// TwinCAT 3 PLC project TcBase
// Title: TcBase
// Company: TcBase
// Author: Giang Nguyen
// ProjectVersion: 0.1.2
// Description: Base library providing basic framework and design patterns.
// ProgramVersion: 3.1.4023.0
// libraries:
//   Base Interfaces,newest,System
//   Tc2_Standard, * (Beckhoff Automation GmbH)
//   Tc2_System, * (Beckhoff Automation GmbH)
//   Tc2_Utilities, * (Beckhoff Automation GmbH)
//   Tc3_DynamicMemory, * (Beckhoff Automation GmbH)
//   Tc3_Module, * (Beckhoff Automation GmbH)
//   TcUnit, * (www.tcunit.org)
// project tree:
//   Action/ FB_Action.TcPOU, FB_RunCyclicTasksAction.TcPOU, I_Action.TcIO
//   Action/Tests/ FB_ActionTestObject.TcPOU, FB_Action_Test.TcPOU, FB_ActivateAction.TcPOU
//   Collection/ FB_List.TcPOU, I_Collection.TcIO, I_Enumerable.TcIO, I_List.TcIO, Param_List.TcGVL
//   Collection/Tests/ FB_ListCapacity_Test.TcPOU, FB_List_Test.TcPOU
//   Context/ FB_Context.TcPOU, I_Context.TcIO
//   Cyclic Task/ I_CyclicTask.TcIO
//   / GVL_IntegerTypeBounds.TcGVL, TestTask.TcTTO
//   Helpers/ F_CompareObjects.TcPOU
//   Invocation Control/ FB_InvocationControl.TcPOU
//   Invocation Control/Tests/ FB_InvocationControlTestTask.TcPOU, FB_InvocationControl_Test.TcPOU
//   Object/ FB_LinkedObject.TcPOU, FB_Object.TcPOU, I_LinkedObject.TcIO, I_Object.TcIO
//   Object/Tests/ FB_DummyObject.TcPOU, FB_Object_Test.TcPOU
//   Observer Pattern/Abstraction/Actions/ FB_NotifyObserverAction.TcPOU
//   Observer Pattern/Abstraction/ FB_AbstractObservable.TcPOU, FB_AbstractObserver.TcPOU, I_Observable.TcIO, I_Observer.TcIO
//   Observer Pattern/ FB_Observable_BOOL.TcPOU, FB_Observable_LINT.TcPOU, FB_Observable_ULINT.TcPOU, FB_Observable_SINT.TcPOU, FB_Observable_DINT.TcPOU, FB_Observable_LWORD.TcPOU, FB_Observable_LREAL.TcPOU, FB_Observable_REAL.TcPOU, FB_Observable_INT.TcPOU, FB_Observable_USINT.TcPOU, FB_Observable_UDINT.TcPOU, FB_Observable_DWORD.TcPOU, FB_Observable_UINT.TcPOU, FB_Observable_BYTE.TcPOU, FB_Observable_WORD.TcPOU, FB_ObserverExt.TcPOU, FB_Observer_LINT.TcPOU, FB_Observer_ULINT.TcPOU, FB_Observer_SINT.TcPOU, FB_Observer_DINT.TcPOU, FB_Observer_LWORD.TcPOU, FB_Observer_LREAL.TcPOU, FB_Observer_REAL.TcPOU, FB_Observer_INT.TcPOU, FB_Observer_USINT.TcPOU, FB_Observer_UDINT.TcPOU, FB_Observer_DWORD.TcPOU, FB_Observer_UINT.TcPOU, FB_Observer_BOOL.TcPOU, FB_Observer_BYTE.TcPOU, FB_Observer_WORD.TcPOU
//   Observer Pattern/Tests/ FB_ObserverPattern_Test.TcPOU, FB_Observer_LREAL_.TcPOU
//   Programs/ Test.TcPOU
//   Restorable/ I_ObjectRestorer.TcIO, I_Restorable.TcIO
//   State Pattern/ FB_State.TcPOU, FB_StateMachine.TcPOU, I_State.TcIO, I_StateMachine.TcIO
//   State Pattern/Tests/ FB_StatePattern_Test.TcPOU
//   State Pattern/Tests/Test Subjects/ E_Season.TcDUT, FB_Autumn.TcPOU, FB_Default.TcPOU, FB_SeasonBase.TcPOU, FB_SeasonStateMachine.TcPOU, FB_Spring.TcPOU, FB_State1.TcPOU, FB_State2.TcPOU, FB_State3.TcPOU, FB_State4.TcPOU, FB_StateMachine1.TcPOU, FB_Summer.TcPOU, FB_Winter.TcPOU, FB_Year.TcPOU, I_SeasonControl.TcIO, I_SeasonState.TcIO
//   Task/Data Type/ E_TaskState.TcDUT
//   Task/ FB_Task.TcPOU, I_Task.TcIO, I_TaskStatus.TcIO

CONFIGURATION TcBase
    RESOURCE PLC ON TwinCAT3
        TASK TestTask(INTERVAL := T#10ms, PRIORITY := 1);
        PROGRAM Test WITH TestTask : Test;
    END_RESOURCE
END_CONFIGURATION

// ---- State Pattern/Tests/Test Subjects/E_Season.TcDUT
{attribute 'qualified_only'}
{attribute 'strict'}
{attribute 'to_string'}
TYPE E_Season :
(
    Autumn,
    Winter,
    Spring,
    Summer
);
END_TYPE

// ---- Task/Data Type/E_TaskState.TcDUT
{attribute 'qualified_only'}
{attribute 'strict'}
{attribute 'to_string'}
TYPE E_TaskState :
(
    Ready := 0,
    Busy,
    Error,
    Done
);
END_TYPE

// ---- Collection/Param_List.TcGVL
{attribute 'qualified_only'}
VAR_GLOBAL CONSTANT
    nDefaultCapacity: UDINT := 4;
    nMaxLength: UDINT := 16#7FEFFFFF;
END_VAR

// ---- GVL_IntegerTypeBounds.TcGVL
{attribute 'qualified_only'}
VAR_GLOBAL CONSTANT
    BYTE_UPPER_BOUND:       BYTE := 16#FF;
    WORD_UPPER_BOUND:       WORD := 16#FFFF;
    DWORD_UPPER_BOUND:      DWORD := 16#FFFF_FFFF;
    LWORD_UPPER_BOUND:      LWORD := 16#FFFF_FFFF_FFFF_FFFF;
    SINT_LOWER_BOUND:       SINT := TO_SINT(16#80);
    SINT_UPPER_BOUND:       SINT := 16#7F;
    USINT_UPPER_BOUND:      USINT := 16#FF;
    INT_LOWER_BOUND:        INT := TO_INT(16#8000);
    INT_UPPER_FOUND:        INT := 16#7FFF;
    UINT_UPPER_BOUND:       UINT := 16#FFFF;
    DINT_LOWER_BOUND:       DINT := TO_DINT(16#8000_0000);
    DINT_UPPER_BOUND:       DINT := 16#7FFF_FFFF;
    UDINT_UPPER_BOUND:      UDINT := 16#FFFF_FFFF;
    LINT_LOWER_BOUND:       LINT := TO_LINT(16#8000_0000_0000_0000);
    LINT_UPPER_BOUND:       LINT := 16#7FFF_FFFF_FFFF_FFFF;
    ULINT_UPPER_BOUND:      ULINT := 16#FFFF_FFFF_FFFF_FFFF;
END_VAR

// ---- Action/I_Action.TcIO
INTERFACE I_Action EXTENDS I_Object

METHOD Execute
VAR_INPUT
    ipObject: I_Object;
END_VAR
END_METHOD

END_INTERFACE

// ---- Collection/I_Collection.TcIO
INTERFACE I_Collection EXTENDS I_Enumerable

METHOD AddItem : DINT
// Returns the index to which the new object is added into the list,
// or -1  to indicate that the object was not inserted
VAR_INPUT
    ipObject:       I_Object;
END_VAR
END_METHOD

METHOD Clear
// Remove all items from the list
VAR_INPUT
END_VAR
END_METHOD

METHOD Contains : BOOL
// Determines whether the list contains the querried object
VAR_INPUT
    ipObject:       I_Object;
END_VAR
END_METHOD

METHOD CopyToArray : BOOL
// Copies the whole list to a compatible one-dimensional array,
// starting at a specified index
VAR_IN_OUT
    aDest:          ARRAY [*] OF I_Object;
END_VAR
VAR_INPUT
    nIdx:           DINT;
END_VAR
END_METHOD

PROPERTY nCount : UDINT
GET
END_GET
END_PROPERTY

METHOD Remove : BOOL
// Remove the first occurerence of a specific object from the list
VAR_INPUT
    ipObject:       I_Object;
END_VAR
END_METHOD

END_INTERFACE

// ---- Collection/I_Enumerable.TcIO
INTERFACE I_Enumerable EXTENDS I_Object

METHOD ForEach : I_Enumerable
VAR_INPUT
    ipAction: I_Action;
END_VAR
END_METHOD

END_INTERFACE

// ---- Collection/I_List.TcIO
INTERFACE I_List EXTENDS I_Collection, I_Enumerable

METHOD IndexOfItem : DINT
// Returns the zero-based index of the object if it was found in the list,
// otherwise returns -1
VAR_INPUT
    ipObject:       I_Object;
END_VAR
END_METHOD

METHOD Insert : BOOL
// Returns TRUE when object is inserted successfully, and FALSE otherwise
VAR_INPUT
    nIdx:       DINT; // Zero-based index at which object should be inserted
    ipObject:   I_Object; // Object to be inserted
END_VAR
END_METHOD

METHOD ItemAt : I_Object
VAR_INPUT
    nIdx:       DINT;
END_VAR
END_METHOD

METHOD LastIndexOf : DINT
VAR_INPUT
    ipObject:       I_Object;
END_VAR
END_METHOD

PROPERTY nCount : UDINT
GET
END_GET
END_PROPERTY

PROPERTY nItemSize : UDINT // Byte-size of each item
GET
END_GET
END_PROPERTY

METHOD RemoveAt : BOOL
// Remove an object at the specified index
VAR_INPUT
    nIdx:       DINT;
END_VAR
END_METHOD

END_INTERFACE

// ---- Context/I_Context.TcIO
INTERFACE I_Context EXTENDS I_Object

END_INTERFACE

// ---- Cyclic Task/I_CyclicTask.TcIO
INTERFACE I_CyclicTask EXTENDS __SYSTEM.IQueryInterface

METHOD Run
VAR_INPUT
END_VAR
END_METHOD

END_INTERFACE

// ---- Object/I_LinkedObject.TcIO
INTERFACE I_LinkedObject EXTENDS I_Object

PROPERTY ipContext : I_Context
GET
END_GET
END_PROPERTY

PROPERTY ipParent : I_LinkedObject
GET
END_GET
END_PROPERTY

END_INTERFACE

// ---- Object/I_Object.TcIO
INTERFACE I_Object EXTENDS __SYSTEM.IQueryInterface

METHOD Equals : BOOL
VAR_INPUT
    ipObject:       I_Object;
END_VAR
END_METHOD

PROPERTY nIdentity : ULINT
GET
END_GET
END_PROPERTY

PROPERTY sPath : STRING(MAX_STRING_LENGTH)
GET
END_GET
END_PROPERTY

END_INTERFACE

// ---- Observer Pattern/Abstraction/I_Observable.TcIO
INTERFACE I_Observable EXTENDS I_Object

METHOD Attach : BOOL
VAR_INPUT
    ipObserver:         I_Observer;
END_VAR
END_METHOD

(*Notify automatically on write access of observable value*)
PROPERTY bAutoNotify : BOOL
GET
END_GET
SET
END_SET
END_PROPERTY

(*Notify only when the value is actually changed*)
PROPERTY bNotifyWhenChanged : BOOL
GET
END_GET
SET
END_SET
END_PROPERTY

METHOD Detach : BOOL
VAR_INPUT
    ipObserver:         I_Observer;
END_VAR
END_METHOD

PROPERTY nDataSize : UDINT
GET
END_GET
END_PROPERTY

PROPERTY nObserverCount : UDINT
GET
END_GET
END_PROPERTY

METHOD NotifyAll : I_Observable
VAR_INPUT
END_VAR
END_METHOD

METHOD NotifyLast : I_Observable
VAR_INPUT
END_VAR
END_METHOD

PROPERTY nTypeClass : __SYSTEM.TYPE_CLASS
GET
END_GET
END_PROPERTY

METHOD ABSTRACT ValueChanged : BOOL
VAR_INPUT
END_VAR
END_METHOD

END_INTERFACE

// ---- Observer Pattern/Abstraction/I_Observer.TcIO
INTERFACE I_Observer EXTENDS I_Object

PROPERTY nTypeClass : __SYSTEM.TYPE_CLASS
GET
END_GET
END_PROPERTY

METHOD Update
VAR_INPUT
    anyVal:         ANY;
END_VAR
END_METHOD

METHOD UpdateP
VAR_INPUT
    pData:          POINTER TO BYTE;
    nTypeClass:     __SYSTEM.TYPE_CLASS;
    nSize:          UDINT;
END_VAR
END_METHOD

END_INTERFACE

// ---- Restorable/I_ObjectRestorer.TcIO
INTERFACE I_ObjectRestorer EXTENDS __SYSTEM.IQueryInterface

METHOD RestoreObject : I_ObjectRestorer
VAR_INPUT
    ipRestorable:           I_Restorable;
END_VAR
END_METHOD

END_INTERFACE

// ---- Restorable/I_Restorable.TcIO
INTERFACE I_Restorable EXTENDS __SYSTEM.IQueryInterface

METHOD Restore : I_Restorable
VAR_INPUT
END_VAR
END_METHOD

END_INTERFACE

// ---- State Pattern/I_State.TcIO
INTERFACE I_State EXTENDS I_Object, I_CyclicTask, I_Restorable

METHOD AssignStateMachine : BOOL
VAR_INPUT
    ipStateMachine:     I_StateMachine;
END_VAR
END_METHOD

PROPERTY ipStateMachine : I_StateMachine
GET
END_GET
END_PROPERTY

METHOD MakeOrphan
VAR_INPUT
END_VAR
END_METHOD

METHOD OnEntry
VAR_INPUT
END_VAR
END_METHOD

METHOD OnExit
VAR_INPUT
END_VAR
END_METHOD

END_INTERFACE

// ---- State Pattern/I_StateMachine.TcIO
INTERFACE I_StateMachine EXTENDS I_Object, I_CyclicTask, I_Restorable

METHOD AddState : BOOL
VAR_INPUT
    ipState:        I_State;
END_VAR
END_METHOD

METHOD ClearStates
VAR_INPUT
END_VAR
END_METHOD

METHOD Contains : BOOL
VAR_INPUT
    ipState:        I_State;
END_VAR
END_METHOD

PROPERTY ipPrevState : I_State
GET
END_GET
END_PROPERTY

PROPERTY ipState : I_State
GET
END_GET
END_PROPERTY

PROPERTY nStateCount : UDINT
GET
END_GET
END_PROPERTY

METHOD SetState : BOOL
VAR_INPUT
    newState:           I_State;
END_VAR
END_METHOD

METHOD StateAt : I_State
VAR_INPUT
    nIdx:       DINT; // Zero-based index to list of state
END_VAR
END_METHOD

END_INTERFACE

// ---- State Pattern/Tests/Test Subjects/I_SeasonControl.TcIO
INTERFACE INTERNAL I_SeasonControl EXTENDS __SYSTEM.IQueryInterface

PROPERTY StateAutumn : I_State
GET
END_GET
END_PROPERTY

PROPERTY StateSpring : I_State
GET
END_GET
END_PROPERTY

PROPERTY StateSummer : I_State
GET
END_GET
END_PROPERTY

PROPERTY StateWinter : I_State
GET
END_GET
END_PROPERTY

END_INTERFACE

// ---- State Pattern/Tests/Test Subjects/I_SeasonState.TcIO
INTERFACE INTERNAL I_SeasonState EXTENDS I_State

PROPERTY bRaining : BOOL
GET
END_GET
END_PROPERTY

PROPERTY bSnowing : BOOL
GET
END_GET
END_PROPERTY

PROPERTY bSunShining : BOOL
GET
END_GET
END_PROPERTY

PROPERTY bWindBlowing : BOOL
GET
END_GET
END_PROPERTY

METHOD ChangeToSummerTyres
VAR_INPUT
END_VAR
END_METHOD

METHOD ChangeToWinterTyres
VAR_INPUT
END_VAR
END_METHOD

PROPERTY eState : E_Season
GET
END_GET
END_PROPERTY

METHOD ABSTRACT NextSeason
VAR_INPUT
END_VAR
END_METHOD

PROPERTY nLeavesState : BYTE
GET
END_GET
END_PROPERTY

PROPERTY nTyresType : BYTE
GET
END_GET
END_PROPERTY

PROPERTY sState : STRING(MAX_STRING_LENGTH)
GET
END_GET
END_PROPERTY

END_INTERFACE

// ---- Task/I_Task.TcIO
INTERFACE I_Task EXTENDS I_Object, I_TaskStatus, I_Restorable

METHOD Abort : I_TaskStatus
VAR_INPUT
END_VAR
END_METHOD

METHOD Invoke : I_TaskStatus
VAR_INPUT
END_VAR
END_METHOD

END_INTERFACE

// ---- Task/I_TaskStatus.TcIO
INTERFACE I_TaskStatus EXTENDS __SYSTEM.IQueryInterface

PROPERTY bBusy : BOOL
GET
END_GET
END_PROPERTY

PROPERTY bDone : BOOL
GET
END_GET
END_PROPERTY

PROPERTY bError : BOOL
GET
END_GET
END_PROPERTY

PROPERTY bReady : BOOL
GET
END_GET
END_PROPERTY

END_INTERFACE

// ---- Programs/Test.TcPOU
PROGRAM Test
VAR
    fbObjectTest: FB_Object_Test;
    fbListTest: FB_List_Test;
    fbListEnsureCapacityTest: FB_ListCapacity_Test;
    fbCallCtrlTest: FB_InvocationControl_Test;
    fbObserverPatternTest: FB_ObserverPattern_Test;
    fbStatePatternTest: FB_StatePattern_Test;
    fbActionTest: FB_Action_Test;
END_VAR

TcUnit.RUN();

END_PROGRAM

// ---- Object/Tests/FB_Object_Test.TcPOU
{attribute 'reflection'}
FUNCTION_BLOCK INTERNAL FB_Object_Test EXTENDS TcUnit.FB_TestSuite
VAR
    fbPathTester: FB_DummyObject;
    _sTestPath: STRING(MAX_STRING_LENGTH) := CONCAT(_sPath, '.fbPathTester');

    {attribute 'instance-path'}
    {attribute 'noinit'}
    _sPath: STRING(MAX_STRING_LENGTH);
END_VAR

TestCompareObjectToSelfExpectTrue();
TestCompareTwoDifferentObjectsExpectFalse();
TestIdentityCorrectness();
TestPathCorrectness();

METHOD PRIVATE TestCompareObjectToSelfExpectTrue
VAR_INST
    fbObject1:      FB_DummyObject;
END_VAR
TcUnit.TEST('TestCompareObjectToSelfExpectTrue');

THIS^.AssertTrue(Condition := fbObject1.Equals(fbObject1),
                 Message := 'Failed when comparing two equal objects');

TcUnit.TEST_FINISHED();
END_METHOD

METHOD PRIVATE TestCompareTwoDifferentObjectsExpectFalse
VAR_INST
    fbObject1:      FB_DummyObject;
    fbObject2:      FB_DummyObject;
END_VAR
TcUnit.TEST('TestCompareTwoDifferentObjectsExpectFalse');

THIS^.AssertFalse(Condition := fbObject1.Equals(fbObject2),
                  Message := 'Failed when comparing two equal objects');

TcUnit.TEST_FINISHED();
END_METHOD

METHOD PRIVATE TestIdentityCorrectness
VAR_INST
    fbObject: FB_DummyObject;
END_VAR
TcUnit.TEST('TestIdentityCorrectness');

THIS^.AssertEquals_ULINT(Expected := ADR(fbObject),
                         Actual := fbObject.nIdentity,
                         Message := 'Object indentity is not true');

TcUnit.TEST_FINISHED();
END_METHOD

METHOD PRIVATE TestPathCorrectness
TcUnit.TEST('TestPathCorrectness');

THIS^.AssertEquals_STRING(Expected := THIS^._sTestPath,
                          Actual := THIS^.fbPathTester.sPath,
                          Message := 'Object path is not true');

TcUnit.TEST_FINISHED();
END_METHOD

END_FUNCTION_BLOCK

// ---- Object/Tests/FB_DummyObject.TcPOU
FUNCTION_BLOCK INTERNAL FB_DummyObject EXTENDS FB_Object
VAR_INPUT
END_VAR
VAR_OUTPUT
END_VAR
VAR
    _nTest: INT;
END_VAR

PROPERTY nTest : INT
GET
nTest := THIS^._nTest;
END_GET
SET
THIS^._nTest := nTest;
END_SET
END_PROPERTY

END_FUNCTION_BLOCK

// ---- Object/FB_Object.TcPOU
{attribute 'reflection'}
FUNCTION_BLOCK ABSTRACT FB_Object IMPLEMENTS I_Object
VAR
    _nIdentity:         ULINT;
    _ipSelf:            I_Object;

    {attribute 'instance-path'}
    {attribute 'noinit'}
    _sPath:             STRING(MAX_STRING_LENGTH);
END_VAR

METHOD Equals : BOOL
VAR_INPUT
    ipObject:       I_Object;
END_VAR
THIS^._ipSelf := THIS^;
Equals := ipObject = THIS^._ipSelf;
END_METHOD

METHOD FB_init : BOOL
VAR_INPUT
    bInitRetains:           BOOL; // if TRUE, the retain variables are initialized (warm start / cold start)
    bInCopyCode:            BOOL;  // if TRUE, the instance afterwards gets moved into the copy code (online change)
END_VAR
THIS^._nIdentity := ADR(THIS^);
THIS^._ipSelf := THIS^;
END_METHOD

PROPERTY nIdentity : ULINT
GET
THIS^._nIdentity := ADR(THIS^);
nIdentity := THIS^._nIdentity;
END_GET
END_PROPERTY

PROPERTY sPath : STRING(MAX_STRING_LENGTH)
GET
sPath := THIS^._sPath;
END_GET
END_PROPERTY

END_FUNCTION_BLOCK

// ---- Collection/Tests/FB_List_Test.TcPOU
FUNCTION_BLOCK INTERNAL FB_List_Test EXTENDS TcUnit.FB_TestSuite
VAR
END_VAR

TestAdd5DifferentItemsExpectAll5Added();
TestAdd5TimesSameObjectExpectAll5Copies();
TestAddNullInterfaceExpectNothingAdded();
TestClearEmptyListExpectSuccess();
TestClearNonEmptyListExpectSuccess();
TestContainsAddedObjectsExpectSuccess();
TestContainsNullObjectExpectFailure();
TestContainsNullObjectFromEmptyListExpectFailure();
TestCopyToArrayOfCompatibleSizeExpectSuccess();
TestCopyToArrayOfIncompatibleSizeExpectFailure();
TestCopyToArrayWithInvalidIndexExpectFailure();
TestEmptyListMustHaveNoItem();
TestForEachWithActivateActionExpectSuccess();
TestForEachWithCylicTaskActionExpectSuccess();
TestIndexOfItem();
TestInsertIntoEmptyListExpectSuccess();
TestInsertIntoListOfItemsExpectSuccess();
TestLastIndexOfListOfMixedDuplicatesAndUniques();
TestRemoveByIndexAndReAddItemExpectCorrectItemOrder();
TestRemoveByIndexFromEmptyListExpectFailure();
TestRemoveByIndexFromListOf5DifferentItemsExpectSuccess();
TestRemoveByIndexFromListOf5ItemsExpectConsistentContents();
TestRemoveByInvalidIndexFromListOfItemsExpectFailure();
TestRemoveInvalidItemFromListExpectFailure();
TestRemoveValidItemFromListExpectSuccess();
TestMeasureAddPerformanceWithVeryManyItemsAdded();

METHOD PRIVATE TestAdd5DifferentItemsExpectAll5Added
VAR_INST
    fbList: FB_List(0);

    aObject: ARRAY [1..5] OF FB_DummyObject;
    ipTmp: I_Object;
    ipCmp: I_Object;
    i: UDINT;
END_VAR
TcUnit.TEST('TestAdd5DifferentItemsExpectAll5Added');

FOR i := 1 TO SIZEOF(aObject)/SIZEOF(aObject[1]) DO
    THIS^.AssertEquals_DINT(Expected := TO_DINT(i - 1),
                            Actual := fbList.AddItem(aObject[i]),
                            Message := 'Failed to add object to list');
END_FOR

THIS^.AssertEquals_UDINT(Expected := SIZEOF(aObject)/SIZEOF(aObject[1]),
                         Actual := fbList.nCount,
                         Message := 'Unexpected number of items added to list');

FOR i := 1 TO SIZEOF(aObject)/SIZEOF(aObject[1]) DO
    ipTmp := fbList.ItemAt(TO_DINT(i - 1));
    ipCmp := aObject[i];
    THIS^.AssertTrue(Condition := ipTmp = ipCmp,
                     Message := CONCAT('Unexpected item at index ', TO_STRING(i)));
END_FOR

TcUnit.TEST_FINISHED();
END_METHOD

METHOD PRIVATE TestAdd5TimesSameObjectExpectAll5Copies
VAR_INST
    fbList: FB_List(0);

    nTimesToAdd: UDINT;
    fbObject: FB_DummyObject;
    ipTmp: I_Object;
    ipCmp: I_Object;
    i: UDINT;
END_VAR
TcUnit.TEST('TestAdd5TimesSameObjectExpectAll5Copies');

nTimesToAdd := 5;

FOR i := 1 TO nTimesToAdd DO
    THIS^.AssertEquals_DINT(Expected := TO_DINT(i - 1),
                            Actual := fbList.AddItem(fbObject),
                            Message := 'Failed to add object to list');
END_FOR

THIS^.AssertEquals_UDINT(Expected := nTimesToAdd,
                         Actual := fbList.nCount,
                         Message := 'Unexpected number of items added to list');

FOR i := 1 TO nTimesToAdd DO
    ipTmp := fbList.ItemAt(TO_DINT(i - 1));
    ipCmp := fbObject;
    THIS^.AssertTrue(Condition := ipTmp = ipCmp,
                     Message := 'Unexpected item added to list');
END_FOR

TcUnit.TEST_FINISHED();
END_METHOD

METHOD PRIVATE TestAddNullInterfaceExpectNothingAdded
VAR_INST
    fbList: FB_List(0);

    ipTmp: I_Object;
    i: UDINT;
END_VAR
TcUnit.TEST('TestAddNullInterfaceExpectNothingAdded');

FOR i := 1 TO 5 DO
    THIS^.AssertEquals_DINT(Expected := -1,
                            Actual := fbList.AddItem(ipTmp),
                            Message := 'Null item added to list');
END_FOR

THIS^.AssertEquals_UDINT(Expected := 0,
                         Actual := fbList.nCount,
                         Message := 'List has item(s) in it, but it should not');

TcUnit.TEST_FINISHED();
END_METHOD

METHOD PRIVATE TestClearEmptyListExpectSuccess
VAR_INST
    fbList: FB_List(0);
END_VAR
TcUnit.TEST('TestClearEmptyListExpectSuccess');

fbList.Clear();

THIS^.AssertEquals_UDINT(Expected := 0,
                         Actual := fbList.nCount,
                         Message := 'List should be empty');

TcUnit.TEST_FINISHED();
END_METHOD

METHOD PRIVATE TestClearNonEmptyListExpectSuccess
VAR_INST
    fbList: FB_List(0);

    aObject: ARRAY [1..5] OF FB_DummyObject;
    ipTmp: I_Object;
    i: UDINT;
END_VAR
TcUnit.TEST('TestClearNonEmptyListExpectSuccess');

FOR i := 1 TO SIZEOF(aObject)/SIZEOF(aObject[1]) DO
    fbList.AddItem(aObject[i]);
END_FOR

THIS^.AssertEquals_UDINT(Expected := SIZEOF(aObject)/SIZEOF(aObject[1]),
                         Actual := fbList.nCount,
                         Message := 'Unexpected number of items added to list');

fbList.Clear();

THIS^.AssertEquals_UDINT(Expected := 0,
                         Actual := fbList.nCount,
                         Message := 'List was not correctly cleared');

FOR i := 1 TO SIZEOF(aObject)/SIZEOF(aObject[1]) DO
    ipTmp := fbList.ItemAt(TO_DINT(i));
    THIS^.AssertTrue(Condition := ipTmp = 0,
                     Message := 'List was not correctly cleared');
END_FOR

TcUnit.TEST_FINISHED();
END_METHOD

METHOD PRIVATE TestContainsAddedObjectsExpectSuccess
VAR_INST
    fbList: FB_List(0);

    aObject: ARRAY [1..5] OF FB_DummyObject;

    ipNull: I_Object;
    i: UDINT;
END_VAR
TcUnit.TEST('TestContainsAddedObjectsExpectSuccess');

FOR i := 1 TO SIZEOF(aObject)/SIZEOF(aObject[1]) DO
    fbList.AddItem(aObject[i]);
END_FOR

FOR i := 1 TO SIZEOF(aObject)/SIZEOF(aObject[1]) DO
    THIS^.AssertTrue(Condition := fbList.Contains(aObject[i]),
                     Message := 'List does not contain added item');
END_FOR

THIS^.AssertFalse(Condition := fbList.Contains(ipNull),
                  Message := 'List should not contain null object');

TcUnit.TEST_FINISHED();
END_METHOD

METHOD PRIVATE TestContainsNullObjectExpectFailure
VAR_INST
    fbList: FB_List(0);

    ipNull: I_Object;
END_VAR
TcUnit.TEST('TestContainsNullObjectExpectFailure');

THIS^.AssertFalse(Condition := fbList.Contains(ipNull),
                  Message := 'List should not contain null object');

TcUnit.TEST_FINISHED();
END_METHOD

METHOD PRIVATE TestContainsNullObjectFromEmptyListExpectFailure
VAR_INST
    fbList: FB_List(0);

    aObject: ARRAY [1..5] OF FB_DummyObject;

    ipNull: I_Object;
    i: UDINT;
END_VAR
TcUnit.TEST('TestContainsNullObjectFromEmptyListExpectFailure');

FOR i := 1 TO SIZEOF(aObject)/SIZEOF(aObject[1]) DO
    fbList.AddItem(aObject[i]);
END_FOR

THIS^.AssertFalse(Condition := fbList.Contains(ipNull),
                  Message := 'List should not contain null object');

TcUnit.TEST_FINISHED();
END_METHOD

METHOD PRIVATE TestCopyToArrayOfCompatibleSizeExpectSuccess
VAR_INST
    fbList: FB_List(0);
    nObjectCount: UDINT;
    aSrcObject: ARRAY [1..10] OF FB_DummyObject;
    aDestObject: ARRAY [1..10] OF I_Object;
    aDestObject2: ARRAY [1..30] OF I_Object;
    i: UDINT;
    ipObject: I_Object;

END_VAR
TcUnit.TEST('TestCopyToArrayOfCompatibleSizeExpectSuccess');

nObjectCount := SIZEOF(aSrcObject)/SIZEOF(aSrcObject[1]);
FOR i := 1 TO nObjectCount DO
    fbList.AddItem(aSrcObject[i]);
END_FOR

// Copy to same size array without offset
THIS^.AssertTrue(Condition := fbList.CopyToArray(aDestObject, 1),
                 Message := 'Failed to copy list to array of same size');

FOR i := 1 TO nObjectCount DO
    ipObject := aSrcObject[i];
    THIS^.AssertTrue(Condition := ipObject = aDestObject[i],
                     Message := 'Expected the same object after in array after copying from list');
END_FOR

// Copy to bigger array with offset
THIS^.AssertTrue(Condition := fbList.CopyToArray(aDestObject2, 14),
                 Message := 'Failed to copy list to array with bigger size');

FOR i := 1 TO nObjectCount DO
    ipObject := aSrcObject[i];
    THIS^.AssertTrue(Condition := ipObject = aDestObject2[i + 13],
                     Message := 'Expected the same object after in array after copying from list');
END_FOR

TcUnit.TEST_FINISHED();
END_METHOD

METHOD PRIVATE TestCopyToArrayOfIncompatibleSizeExpectFailure
VAR_INST
    fbList: FB_List(0);
    nObjectCount: UDINT;
    aSrcObject: ARRAY [1..10] OF FB_DummyObject;
    aDestObject: ARRAY [1..5] OF I_Object;
    i: UDINT;
END_VAR
TcUnit.TEST('TestCopyToArrayOfIncompatibleSizeExpectFailure');

nObjectCount := SIZEOF(aSrcObject)/SIZEOF(aSrcObject[1]);
FOR i := 1 TO nObjectCount DO
    fbList.AddItem(aSrcObject[i]);
END_FOR

THIS^.AssertFalse(Condition := fbList.CopyToArray(aDestObject, 1),
                  Message := 'Failed to copy list to array of same size');

FOR i := 1 TO SIZEOF(aDestObject)/SIZEOF(aDestObject[1]) DO
    THIS^.AssertTrue(Condition := aDestObject[i] = 0,
                     Message := 'Array should be "empty" after copying due to being smaller than list');
END_FOR

TcUnit.TEST_FINISHED();
END_METHOD

METHOD PRIVATE TestCopyToArrayWithInvalidIndexExpectFailure
VAR_INST
    fbList: FB_List(0);
    nObjectCount: UDINT;
    aSrcObject: ARRAY [1..10] OF FB_DummyObject;
    aDestObject: ARRAY [1..10] OF I_Object;
    aDestObject2: ARRAY [1..30] OF I_Object;
    i: UDINT;

END_VAR
TcUnit.TEST('TestCopyToArrayWithInvalidIndexExpectFailure');

nObjectCount := SIZEOF(aSrcObject)/SIZEOF(aSrcObject[1]);
FOR i := 1 TO nObjectCount DO
    fbList.AddItem(aSrcObject[i]);
END_FOR

// Copy to same size array
THIS^.AssertFalse(Condition := fbList.CopyToArray(aDestObject, 2),
                  Message := 'List should not copy items to array using invalid index');

FOR i := 1 TO nObjectCount DO
    THIS^.AssertTrue(Condition := 0 = aDestObject[i],
                     Message := 'Array should be "empty" after copying due to being smaller than list');
END_FOR

// Copy to bigger array
THIS^.AssertFalse(Condition := fbList.CopyToArray(aDestObject2, 22),
                  Message := 'List should not copy items to array using invalid index');

FOR i := 1 TO nObjectCount DO
    THIS^.AssertTrue(Condition := 0 = aDestObject2[i + 13],
                     Message := 'Array should be "empty" after copying due to being smaller than list');
END_FOR

THIS^.AssertFalse(Condition := fbList.CopyToArray(aDestObject2, 0),
                  Message := 'List should not copy items to array using invalid index');

FOR i := 1 TO nObjectCount DO
    THIS^.AssertTrue(Condition := 0 = aDestObject2[i + 13],
                     Message := 'Array should be "empty" after copying due to being smaller than list');
END_FOR

TcUnit.TEST_FINISHED();
END_METHOD

METHOD PRIVATE TestEmptyListMustHaveNoItem
VAR_INST
    fbList:     FB_List(0);
END_VAR
TcUnit.TEST('TestEmptyListMustHaveNoItem');

THIS^.AssertEquals_UDINT(Expected := 0,
                         Actual := fbList.nCount,
                         Message := 'Empty list must not have any item(s)');

TcUnit.TEST_FINISHED();
END_METHOD

METHOD PRIVATE TestForEachWithActivateActionExpectSuccess
VAR_INST
    i: UDINT;
    fbList: FB_List(0);
    aObject: ARRAY [1..10] OF FB_ActionTestObject;
    fbActivateObjects: FB_ActivateAction;
END_VAR
TcUnit.TEST('TestForEachWithActivateActionExpectSuccess');

FOR i := 1 TO SIZEOF(aObject)/SIZEOF(aObject[1]) DO
    fbList.AddItem(aObject[i]);
END_FOR

fbList.ForEach(fbActivateObjects.Inputs(TRUE));

FOR i := 1 TO SIZEOF(aObject)/SIZEOF(aObject[1]) DO
     THIS^.AssertTrue(Condition := aObject[1].bIsActivated,
                      Message := 'Failed to activate object(s)');
END_FOR

TcUnit.TEST_FINISHED();
END_METHOD

METHOD PRIVATE TestForEachWithCylicTaskActionExpectSuccess
VAR_INST
    nCyclesToRun: UDINT := 5;
    nCounter: UDINT := 0;
    i: UDINT;
    fbList: FB_List(0);
    aObject: ARRAY [1..10] OF FB_ActionTestObject;
    fbRunCyclicTask: FB_RunCyclicTasksAction;
END_VAR
TcUnit.TEST('TestForEachWithCylicTaskActionExpectSuccess');

IF nCounter = 0 THEN
    FOR i := 1 TO SIZEOF(aObject)/SIZEOF(aObject[1]) DO
        fbList.AddItem(aObject[i]);
    END_FOR
END_IF

fbList.ForEach(fbRunCyclicTask);
nCounter := nCounter + 1;

IF nCyclesToRun = nCounter THEN
    FOR i := 1 TO SIZEOF(aObject)/SIZEOF(aObject[1]) DO
        THIS^.AssertEquals_UDINT(Expected := nCyclesToRun,
                                 Actual := aObject[i].nCounter,
                                 Message := 'Unexpected counter value of cyclic object');
    END_FOR
    TcUnit.TEST_FINISHED();
END_IF
END_METHOD

METHOD PRIVATE TestIndexOfItem
VAR_INST
    fbList: FB_List(0);

    aObject: ARRAY [1..10] OF FB_DummyObject;
    fbObject1: FB_DummyObject;
    fbObject2: FB_DummyObject;
    fbObject3: FB_DummyObject;

    ipNull: I_Object;
    i: UDINT;
END_VAR
TcUnit.TEST('TestIndexQuerryCorrectness');

FOR i := 1 TO SIZEOF(aObject)/SIZEOF(aObject[1]) DO
    fbList.AddItem(aObject[i]);
END_FOR

FOR i := 1 TO SIZEOF(aObject)/SIZEOF(aObject[1]) DO
    THIS^.AssertEquals_DINT(Expected := TO_DINT(i - 1),
                            Actual := fbList.IndexOfItem(aObject[i]),
                            Message := 'Unexpected index of added item');
END_FOR

fbList.Clear();

FOR i := 1 TO SIZEOF(aObject)/SIZEOF(aObject[1]) DO
    THIS^.AssertEquals_DINT(Expected := -1,
                            Actual := fbList.IndexOfItem(aObject[i]),
                            Message := 'Item still found from list even though it has been cleared');
END_FOR

THIS^.AssertEquals_DINT(Expected := -1,
                        Actual := fbList.IndexOfItem(ipNull),
                        Message := 'Invalid result when querying index of a null item');

fbList.AddItem(fbObject1);
fbList.AddItem(fbObject3);
fbList.AddItem(fbObject1);
fbList.AddItem(fbObject2);
fbList.AddItem(fbObject2);

THIS^.AssertEquals_DINT(Expected := 0,
                        Actual := fbList.IndexOfItem(fbObject1),
                        Message := 'IndexOfItem() should return the index of the first match if there are multiple copies');
THIS^.AssertEquals_DINT(Expected := 1,
                        Actual := fbList.IndexOfItem(fbObject3),
                        Message := 'IndexOfItem() should return the index of the first match if there are multiple copies');
THIS^.AssertEquals_DINT(Expected := 3,
                        Actual := fbList.IndexOfItem(fbObject2),
                        Message := 'IndexOfItem() should return the index of the first match if there are multiple copies');


TcUnit.TEST_FINISHED();
END_METHOD

METHOD PRIVATE TestInsertIntoEmptyListExpectSuccess
VAR_INST
    fbList: FB_List(0);

    aObject: ARRAY [1..10] OF FB_DummyObject;
    aInsPos: ARRAY [1..10] OF DINT;
    ipTmp: I_Object;
    ipCmp: I_Object;

    i: UDINT;
END_VAR
TcUnit.TEST('TestInsertIntoEmptyListExpectSuccess');

FOR i := 1 TO SIZEOF(aObject)/SIZEOF(aObject[1]) DO
    IF i = 4 THEN
        aInsPos[i] := 0;
    ELSIF i = 8 THEN
        aInsPos[i] := 4;;
    ELSIF i = 10 THEN
        aInsPos[i] := 1;
    ELSE
        aInsPos[i] := TO_DINT(i - 1);
    END_IF

    THIS^.AssertTrue(Condition := fbList.Insert(nIdx := aInsPos[i], aObject[i]),
                     Message := 'Could not insert item to list');

    ipTmp := fbList.ItemAt(aInsPos[i]);
    ipCmp := aObject[i];
    THIS^.AssertTrue(Condition := ipTmp = ipCmp,
                     Message := 'Added item is not at the expected index');
END_FOR

THIS^.AssertEquals_UDINT(Expected := SIZEOF(aObject)/SIZEOF(aObject[1]),
                         Actual := fbList.nCount,
                         Message := 'Unexpected number of items inserted to list');

FOR i := 1 TO SIZEOF(aObject)/SIZEOF(aObject[1]) DO
    THIS^.AssertTrue(Condition := fbList.Contains(aObject[i]),
                     Message := 'List does not contain inserted item');
END_FOR

TcUnit.TEST_FINISHED();
END_METHOD

METHOD PRIVATE TestInsertIntoListOfItemsExpectSuccess
VAR_INST
    fbList: FB_List(0);

    aObject: ARRAY [1..10] OF FB_DummyObject;
    aObjectToInsert: ARRAY [1..3] OF FB_DummyObject;
    aInsPos: ARRAY [1..3] OF DINT;
    ipTmp: I_Object;
    ipCmp: I_Object;

    i: UDINT;
END_VAR
TcUnit.TEST('TestInsertIntoListOfItemsExpectSuccess');

{region "Insert to head, end, and middle"}
FOR i := 1 TO SIZEOF(aObject)/SIZEOF(aObject[1]) DO
    fbList.AddItem(aObject[i]);
END_FOR

aInsPos[1] := 0;
aInsPos[2] := TO_DINT(fbList.nCount + 1);
aInsPos[3] := 3;

FOR i := 1 TO SIZEOF(aInsPos)/SIZEOF(aInsPos[1]) DO
    THIS^.AssertTrue(Condition := fbList.Insert(aInsPos[i], aObjectToInsert[i]),
                     Message := 'Failed to insert item into list');

    ipTmp := fbList.ItemAt(aInsPos[i]);
    ipCmp := aObjectToInsert[i];
    THIS^.AssertTrue(Condition := ipTmp = ipCmp,
                     Message := 'Added item is not at the expected index');
END_FOR

THIS^.AssertEquals_UDINT(Expected := SIZEOF(aObject)/SIZEOF(aObject[1])
                                     + SIZEOF(aObjectToInsert)/SIZEOF(aObjectToInsert[1]),
                         Actual := fbList.nCount,
                         Message := 'Unexpected number of items inserted to list');

FOR i := 1 TO SIZEOF(aObject)/SIZEOF(aObject[1]) DO
    THIS^.AssertTrue(Condition := fbList.Contains(aObject[i]),
                     Message := 'List does not contain inserted item');
END_FOR

FOR i := 1 TO SIZEOF(aObjectToInsert)/SIZEOF(aObjectToInsert[1]) DO
    THIS^.AssertTrue(Condition := fbList.Contains(aObjectToInsert[i]),
                     Message := 'List does not contain inserted item');
END_FOR
{endregion}

fbList.Clear();

{region "Insert to middle"}
FOR i := 1 TO SIZEOF(aObject)/SIZEOF(aObject[1]) DO
    fbList.AddItem(aObject[i]);
END_FOR

aInsPos[1] := 8;
aInsPos[2] := 5;
aInsPos[3] := 1;

FOR i := 1 TO SIZEOF(aInsPos)/SIZEOF(aInsPos[1]) DO
    THIS^.AssertTrue(Condition := fbList.Insert(aInsPos[i], aObjectToInsert[i]),
                     Message := 'Failed to insert item into list');

    ipTmp := fbList.ItemAt(aInsPos[i]);
    ipCmp := aObjectToInsert[i];
    THIS^.AssertTrue(Condition := ipTmp = ipCmp,
                     Message := 'Added item is not at the expected index');
END_FOR

THIS^.AssertEquals_UDINT(Expected := SIZEOF(aObject)/SIZEOF(aObject[1])
                                     + SIZEOF(aObjectToInsert)/SIZEOF(aObjectToInsert[1]),
                         Actual := fbList.nCount,
                         Message := 'Unexpected number of items inserted to list');

FOR i := 1 TO SIZEOF(aObject)/SIZEOF(aObject[1]) DO
    THIS^.AssertTrue(Condition := fbList.Contains(aObject[i]),
                     Message := 'List does not contain inserted item');
END_FOR

FOR i := 1 TO SIZEOF(aObjectToInsert)/SIZEOF(aObjectToInsert[1]) DO
    THIS^.AssertTrue(Condition := fbList.Contains(aObjectToInsert[i]),
                     Message := 'List does not contain inserted item');
END_FOR
{endregion}

TcUnit.TEST_FINISHED();
END_METHOD

METHOD PRIVATE TestLastIndexOfListOfMixedDuplicatesAndUniques
VAR_INST
    fbList: FB_List(0);

    aObject: ARRAY [1..5] OF FB_DummyObject;
    aAddOrder: ARRAY[1..20] OF I_Object;
    aExpLastIdx: ARRAY [1..5] OF DINT;
    nIdx: UDINT;
    nObjectCount: UDINT;
    nTimesToAdd: UDINT;
    i: UDINT;
    fbRand: DRAND := (Seed := 128);
    sMessage: STRING(255);
END_VAR
TcUnit.TEST('TestLastIndexOfListOfMixedDuplicatesAndUniques');

nObjectCount := SIZEOF(aObject)/SIZEOF(aObject[1]);
nTimesToAdd := SIZEOF(aAddOrder)/SIZEOF(aAddOrder[1]);

FOR i := 1 TO nTimesToAdd DO
    fbRand();
    nIdx := TO_UDINT(fbRand.Num*(nObjectCount - 1)) + 1;
    aAddOrder[i] := aObject[nIdx];

    IF aExpLastIdx[nIdx] < TO_DINT(i) THEN
        aExpLastIdx[nIdx] := TO_DINT(i);
    END_IF
END_FOR

FOR i := 1 TO nTimesToAdd DO
    fbList.AddItem(aAddOrder[i]);
END_FOR

FOR i := 1 TO nObjectCount DO
    sMessage := Tc2_Standard.CONCAT('Unexpected last index of object at idx ', TO_STRING(i));
    THIS^.AssertEquals_DINT(Expected := aExpLastIdx[i] - 1,
                            Actual := fbList.LastIndexOf(aObject[i]),
                            Message := sMessage);
END_FOR

TcUnit.TEST_FINISHED();
END_METHOD

METHOD PRIVATE TestMeasureAddPerformanceWithVeryManyItemsAdded
VAR_INST
    fbList: FB_List(0);
    fbObject: FB_DummyObject;
    fbProfiler: Tc2_Utilities.Profiler;

    nTimesToAdd: UDINT := 100000;
    i: UDINT;
    stProfileData: Tc2_Utilities.PROFILERSTRUCT;
    sMsg: STRING(255);
END_VAR
IF TcUnit.TEST_ORDERED('TestMeasureAddPerformanceWithVeryManyItemsAdded') THEN
    IF nTimesToAdd > 0 THEN
        fbProfiler(START := TRUE, RESET := TRUE);
        FOR i := 1 TO nTimesToAdd DO
            fbList.AddItem(fbObject);
        END_FOR

        THIS^.AssertEquals_UDINT(Expected := TO_UDINT(nTimesToAdd),
                                 Actual := fbList.nCount,
                                 Message := 'Unexpected number of items added to list');

        fbProfiler(START := FALSE);
        stProfileData := fbProfiler.DATA;

        sMsg := 'Took ';
        sMsg := CONCAT(sMsg, TO_STRING(stProfileData.LastExecTime));
        sMsg := CONCAT(sMsg, 'us to add ');
        sMsg := CONCAT(sMsg, TO_STRING(nTimesToAdd));
        sMsg := CONCAT(sMsg, ' item(s) to list. ');
        sMsg := CONCAT(sMsg, 'On average ');
        sMsg := CONCAT(sMsg, TO_STRING(TO_LREAL(fbProfiler.DATA.AverageExecTime)/TO_LREAL(nTimesToAdd)));
        sMsg := CONCAT(sMsg, 'us');
        sMsg := CONCAT(sMsg, ' per item');

        Tc2_System.ADSLOGSTR(msgCtrlMask := Tc2_System.ADSLOG_MSGTYPE_ERROR,
                             msgFmtStr := sMsg,
                             strArg := '');
    END_IF

    TcUnit.TEST_FINISHED();
END_IF
END_METHOD

METHOD PRIVATE TestRemoveByIndexAndReAddItemExpectCorrectItemOrder
VAR_INST
    fbList: FB_List(0);
    aObject: ARRAY [1..5] OF FB_DummyObject;
    aIdx: ARRAY [1..5] OF UDINT
        := [3, 2, 4, 5, 1];
    nArraySize: UDINT;
    i: UDINT;
    j: UDINT;
END_VAR
TcUnit.TEST('TestRemoveByIndexAndReAddItemExpectCorrectItemOrder');
nArraySize := SIZEOF(aObject)/SIZEOF(aObject[1]);

FOR i := 1 TO nArraySize DO
    fbList.AddItem(aObject[i]);
END_FOR

FOR i := 1 TO nArraySize DO
    fbList.RemoveAt(fbList.IndexOfItem(aObject[aIdx[i]]));
    fbList.AddItem(aObject[aIdx[i]]);
END_FOR

FOR i := 1 TO nArraySize DO
    THIS^.AssertTrue(Condition := fbList.ItemAt(TO_DINT(i) - 1).Equals(aObject[aIdx[i]]),
                     Message := CONCAT('Unexpected item found at ', TO_STRING(i - 1)));
END_FOR

TcUnit.TEST_FINISHED();
END_METHOD

METHOD PRIVATE TestRemoveByIndexFromEmptyListExpectFailure
VAR_INST
    fbList: FB_List(0);

    aIdx: ARRAY[1..10] OF DINT := 
        [0, 1, 2, 3, 4, 5, 6, 7, 8, 9];

    i: UDINT;
END_VAR
TcUnit.TEST('TestRemoveByIndexFromEmptyListExpectFailure');

FOR i := 1 TO SIZEOF(aIdx)/SIZEOF(aIdx[1]) DO
    THIS^.AssertFalse(Condition := fbList.RemoveAt(aIdx[i]),
                      Message := 'Empty list should not have any item to be removed');
END_FOR

TcUnit.TEST_FINISHED();
END_METHOD

METHOD PRIVATE TestRemoveByIndexFromListOf5DifferentItemsExpectSuccess
VAR_INST
    fbList: FB_List(0);
    aObject: ARRAY [1..5] OF FB_DummyObject;

    nArraySize: UDINT;
    i: UDINT;
END_VAR
TcUnit.TEST('TestRemoveItemFromListOf5DifferentItemsExpectSuccess');
nArraySize := SIZEOF(aObject)/SIZEOF(aObject[1]);

// Remove from last to first
FOR i := 1 TO nArraySize DO
    fbList.AddItem(aObject[i]);
END_FOR

FOR i := 1 TO nArraySize DO
    THIS^.AssertTrue(Condition := fbList.RemoveAt(TO_DINT(nArraySize - i)),
                     Message := 'Could not remove added item');

    THIS^.AssertEquals_UDINT(Expected := nArraySize - i,
                             Actual := fbList.nCount,
                             Message := 'Unexpected number of items after removal');
END_FOR

// Remove from first
FOR i := 1 TO nArraySize DO
    fbList.AddItem(aObject[i]);
END_FOR

FOR i := 1 TO nArraySize DO
    THIS^.AssertTrue(Condition := fbList.RemoveAt(0),
                     Message := 'Could not remove added item');

    THIS^.AssertEquals_UDINT(Expected := nArraySize - i,
                             Actual := fbList.nCount,
                             Message := 'Unexpected number of items after removal');
END_FOR

// Remove from middle to first
FOR i := 1 TO nArraySize DO
    fbList.AddItem(aObject[i]);
END_FOR

FOR i := 1 TO nArraySize DO
    THIS^.AssertTrue(Condition := fbList.RemoveAt(MAX(0, 3 - TO_DINT(i))),
                     Message := 'Could not remove added item');

    THIS^.AssertEquals_UDINT(Expected := nArraySize - i,
                             Actual := fbList.nCount,
                             Message := 'Unexpected number of items after removal');
END_FOR

TcUnit.TEST_FINISHED();
END_METHOD

METHOD PRIVATE TestRemoveByIndexFromListOf5ItemsExpectConsistentContents
VAR_INST
    fbList: FB_List(0);
    aObject: ARRAY [1..5] OF FB_DummyObject;
    nArraySize: UDINT;
    i: UDINT;
    j: UDINT;
END_VAR
TcUnit.TEST('TestRemoveByIndexFromListOf5ItemsExpectConsistentContents');
nArraySize := SIZEOF(aObject)/SIZEOF(aObject[1]);

FOR i := 1 TO nArraySize DO
    fbList.AddItem(aObject[i]);
END_FOR

FOR i := 1 TO nArraySize DO
    fbList.RemoveAt(0);

    // After every removal, we check that the content of the list is correct
    IF fbList.nCount > 0 THEN
        FOR j := 0 TO fbList.nCount - 1 DO
            THIS^.AssertTrue(Condition := fbList.ItemAt(TO_DINT(j)).Equals(aObject[i + j + 1]),
                             Message := 'Unexpected list contents after removing item');
        END_FOR
    END_IF
END_FOR

TcUnit.TEST_FINISHED();
END_METHOD

METHOD PRIVATE TestRemoveByInvalidIndexFromListOfItemsExpectFailure
VAR_INST
    fbList: FB_List(0);

    aIdx: ARRAY[1..10] OF DINT := 
        [-1, 5, 6, 7, 10, -10, -3, -4, -2, 9];
    aObject: ARRAY [1..5] OF FB_DummyObject;

    i: UDINT;
END_VAR
TcUnit.TEST('TestRemoveByInvalidIndexFromListOfItemsExpectFailure');

FOR i := 1 TO SIZEOF(aObject)/SIZEOF(aObject[1]) DO
    fbList.AddItem(aObject[i]);
END_FOR

FOR i := 1 TO SIZEOF(aIdx)/SIZEOF(aIdx[1]) DO
    THIS^.AssertFalse(Condition := fbList.RemoveAt(aIdx[i]),
                      Message := 'Removing item with out-of-bound index should not succeed');
END_FOR

THIS^.AssertEquals_UDINT(Expected := 5,
                         Actual := fbList.nCount,
                         Message := 'Item(s) were successfully removed from list with out-of-bound index');

TcUnit.TEST_FINISHED();
END_METHOD

METHOD PRIVATE TestRemoveInvalidItemFromListExpectFailure
VAR_INST
    fbList: FB_List(0);

    aObject: ARRAY [1..10] OF FB_DummyObject;
    ipNull: I_Object;
    fbObject: FB_DummyObject;

    i: UDINT;
END_VAR
TcUnit.TEST('TestRemoveInvalidItemFromListExpectFailure');

FOR i := 1 TO SIZEOF(aObject)/SIZEOF(aObject[1]) DO
    fbList.AddItem(aObject[i]);
END_FOR

THIS^.AssertFalse(Condition := fbList.Remove(ipNull),
                  Message := 'Unexpectedly removed a null item');

THIS^.AssertFalse(Condition := fbList.Remove(fbObject),
                  Message := 'List should not be able to remove item it does not contain');

THIS^.AssertEquals_UDINT(Expected := SIZEOF(aObject)/SIZEOF(aObject[1]),
                         Actual := fbList.nCount,
                         Message := 'Unexpected number of items after invalid removal');

FOR i := 1 TO SIZEOF(aObject)/SIZEOF(aObject[1]) DO
    THIS^.AssertTrue(Condition := fbList.Remove(aObject[i]),
                     Message := 'Could not remove added item');

    THIS^.AssertFalse(Condition := fbList.Remove(aObject[i]),
                      Message := 'Removed item was unexpectedly removed twice');

    THIS^.AssertEquals_UDINT(Expected := SIZEOF(aObject)/SIZEOF(aObject[1]) - i,
                             Actual := fbList.nCount,
                             Message := 'Unexpected number of items after removal');
END_FOR

TcUnit.TEST_FINISHED();
END_METHOD

METHOD PRIVATE TestRemoveValidItemFromListExpectSuccess
VAR_INST
    fbList: FB_List(0);

    aObject: ARRAY [1..10] OF FB_DummyObject;

    i: UDINT;
END_VAR
TcUnit.TEST('TestRemoveValidItemFromListExpectSuccess');

FOR i := 1 TO SIZEOF(aObject)/SIZEOF(aObject[1]) DO
    fbList.AddItem(aObject[i]);
END_FOR

FOR i := 1 TO SIZEOF(aObject)/SIZEOF(aObject[1]) DO
    THIS^.AssertTrue(Condition := fbList.Remove(aObject[i]),
                     Message := 'Could not remove added item');

    THIS^.AssertEquals_UDINT(Expected := SIZEOF(aObject)/SIZEOF(aObject[1]) - i,
                             Actual := fbList.nCount,
                             Message := 'Unexpected number of items after removal');
END_FOR

TcUnit.TEST_FINISHED();
END_METHOD

END_FUNCTION_BLOCK

// ---- Collection/FB_List.TcPOU
FUNCTION_BLOCK FB_List EXTENDS FB_Object IMPLEMENTS I_List
VAR
    fbMemMan:       FB_DynMem_Manager;
    fbBuffer:       FB_DynMem_Buffer(ipMemMan := fbMemMan);
    _nCount:        UDINT;
END_VAR

METHOD AddItem : DINT
VAR_INPUT
    ipObject:       I_Object;
END_VAR
IF ipObject = 0 THEN
    AddItem := -1;
    RETURN;
END_IF

IF THIS^.IsFull() THEN
    AddItem := -1;
    RETURN;
END_IF

IF THIS^.nCount = THIS^.nCapacity THEN
    THIS^.EnsureCapacity(THIS^.nCount + 1);
END_IF

THIS^._nCount := THIS^._nCount + 1;
THIS^.WriteToBuffer(nIdx := THIS^.nLastIdx, ipObject := ipObject);
AddItem := THIS^.nLastIdx;
END_METHOD

METHOD Clear
THIS^.fbBuffer.Resize(nSize := 0,
                      bPreserve := FALSE,
                      bReset := TRUE);

THIS^._nCount := 0;
END_METHOD

METHOD Contains : BOOL
VAR_INPUT
    ipObject:       I_Object;
END_VAR
VAR
    i:              DINT;
    ipTmp:          I_Object;
END_VAR
IF ipObject = 0 THEN
    RETURN;
END_IF

FOR i := 0 TO THIS^.nLastIdx DO
    IF F_CompareObjects(ipObject, THIS^.ItemAt(i)) THEN
        Contains := TRUE;
        RETURN;
    END_IF
END_FOR
END_METHOD

METHOD CopyToArray : BOOL
// Copies the whole list to a compatible one-dimensional array,
// starting at a specified index
VAR_IN_OUT
    aDest:          ARRAY [*] OF I_Object;
END_VAR
VAR_INPUT
    nIdx:           DINT;
END_VAR
VAR
    nLowerBnd:      DINT;
    nUpperBnd:      DINT;
    i:              DINT;
END_VAR
// Nothing to copy
IF THIS^.nCount = 0 THEN
    RETURN;
END_IF

nLowerBnd := LOWER_BOUND(aDest, 1);
nUpperBnd := UPPER_BOUND(aDest, 1);

// Invalid index given
IF nIdx < nLowerBnd OR_ELSE nUpperBnd < nIdx THEN
    RETURN;
END_IF

// Array not big enough
IF TO_UDINT(nUpperBnd - nIdx + 1) < THIS^.nCount THEN
    RETURN;
END_IF

Tc2_System.MEMCPY(destAddr := ADR(aDest[nIdx]),
                  srcAddr := THIS^.pBuffer,
                  n := THIS^.nCount*THIS^.nItemSize);

CopyToArray := TRUE;
END_METHOD

METHOD PRIVATE EnsureCapacity : BOOL
VAR_INPUT
    nMin: UDINT;
END_VAR
VAR
    nNewCapacity: UDINT;
END_VAR
IF THIS^.nCapacity > nMin THEN
    RETURN;
END_IF

nNewCapacity := SEL(THIS^.nCapacity = 0, THIS^.nCapacity * 2, Param_List.nDefaultCapacity);
nNewCapacity := LIMIT(nMin, nNewCapacity, Param_List.nMaxLength);

EnsureCapacity := THIS^.fbBuffer.Resize(nSize := nNewCapacity*THIS^.nItemSize,
                                        bPreserve := TRUE,
                                        bReset := FALSE);
END_METHOD

METHOD FB_init : BOOL
VAR_INPUT
    bInitRetains:   BOOL; // if TRUE, the retain variables are initialized (warm start / cold start)
    bInCopyCode:    BOOL;  // if TRUE, the instance afterwards gets moved into the copy code (online change)
    nCapacity:      UDINT;
END_VAR
THIS^.fbBuffer.CreateBuffer(nSize := nCapacity*THIS^.nItemSize,
                            bReset := TRUE);
END_METHOD

METHOD ForEach : I_Enumerable
VAR_INPUT
    ipAction: I_Action;
END_VAR
VAR
    i: DINT;
END_VAR
ForEach := THIS^;

IF THIS^.nCount = 0 OR_ELSE ipAction = 0 THEN
    RETURN;
END_IF

FOR i := 0 TO TO_DINT(THIS^.nCount) - 1 DO
    ipAction.Execute(THIS^.ItemAt(i));
END_FOR
END_METHOD

METHOD PRIVATE GetOffset : PVOID
VAR_INPUT
    nIdx: DINT;
END_VAR
VAR
    pTmp: POINTER TO I_Object;
END_VAR
pTmp := THIS^.pBuffer;
GetOffset := ADR(pTmp[nIdx]);
END_METHOD

METHOD PRIVATE IndexIsValid : BOOL
VAR_INPUT
    nIdx:       DINT;
END_VAR
IndexIsValid := (0 <= nIdx) AND_THEN (nIdx <= THIS^.nLastIdx);
END_METHOD

METHOD IndexOfItem : DINT
VAR_INPUT
    ipObject:   I_Object;
END_VAR
VAR
    i:          DINT;
    ipTmp:      I_Object;
END_VAR
IF ipObject = 0 THEN
    IndexOfItem := -1;
    RETURN;
END_IF

FOR i := 0 TO THIS^.nLastIdx DO
    ipTmp := THIS^.ItemAt(i);
    IF F_CompareObjects(ipTmp, ipObject) THEN
        IndexOfItem := i;
        RETURN;
    END_IF
END_FOR

IndexOfItem := -1;
END_METHOD

METHOD Insert : BOOL
VAR_INPUT
    (* Zero-based index at which object should be inserted*)
    nIdx: DINT;
    (* Object to be inserted*)
    ipObject: I_Object;
END_VAR
VAR
    nIdxTmp:    DINT;
END_VAR
IF ipObject = 0
    OR_ELSE THIS^.IsFull() THEN
    RETURN;
END_IF

IF nIdx < 0 THEN
    RETURN;
END_IF

// If given index is larger than (last idx + 1) then limit
// the index so that the item is appended to the end
nIdxTmp := MIN(nIdx, THIS^.nLastIdx + 1);

IF nIdxTmp = (THIS^.nLastIdx + 1) THEN
    Insert := THIS^.AddItem(ipObject) <> -1;
    RETURN;
END_IF

IF THIS^.nCount = THIS^.nCapacity THEN
    THIS^.EnsureCapacity(THIS^.nCount + 1);
END_IF

Tc2_System.MEMMOVE(destAddr := THIS^.GetOffset(nIdx := nIdx + 1),
                   srcAddr := THIS^.GetOffset(nIdx := nIdx),
                   n := TO_UDINT(THIS^.nLastIdx - nIdx + 1)*THIS^.nItemSize);

THIS^.WriteToBuffer(nIdx := nIdx, ipObject := ipObject);
THIS^._nCount := THIS^._nCount + 1;

Insert := TRUE;
END_METHOD

METHOD PROTECTED IsFull : BOOL
VAR_INPUT
END_VAR
IF THIS^.nCount >= TO_UDINT(GVL_IntegerTypeBounds.DINT_UPPER_BOUND) THEN
    IsFull := TRUE;
END_IF
END_METHOD

METHOD ItemAt : I_Object
VAR_INPUT
    nIdx:       DINT;
END_VAR
VAR
    pTmp:       POINTER TO I_Object;
END_VAR
pTmp := THIS^.pBuffer;
IF THIS^.IndexIsValid(nIdx)
    AND_THEN pTmp <> 0 THEN
    ItemAt := pTmp[nIdx];
END_IF
END_METHOD

METHOD LastIndexOf : DINT
VAR_INPUT
    ipObject:       I_Object;
END_VAR
VAR
    i:              UDINT;
    ipTmp:          I_Object;
END_VAR
IF THIS^.nCount = 0
    OR_ELSE ipObject = 0 THEN
    LastIndexOf := -1;
    RETURN;
END_IF

FOR i := 0 TO TO_UDINT(THIS^.nLastIdx) DO
    ipTmp := THIS^.ItemAt(TO_DINT(i));
    IF ipTmp = ipObject THEN
        LastIndexOf := TO_DINT(i);
    END_IF
END_FOR

IF LastIndexOf = 0 THEN
    LastIndexOf := -1;
END_IF
END_METHOD

PROPERTY nCapacity : UDINT
GET
IF THIS^.nItemSize <> 0 THEN
    nCapacity := THIS^.fbBuffer.nBufferSize/THIS^.nItemSize;
END_IF
END_GET
END_PROPERTY

PROPERTY nCount : UDINT
GET
nCount := THIS^._nCount;
END_GET
END_PROPERTY

PROPERTY nItemSize : UDINT
GET
nItemSize := SIZEOF(POINTER TO I_Object);
END_GET
END_PROPERTY

PROPERTY PRIVATE nLastIdx : DINT
GET
IF THIS^.nCount > 0 THEN
    nLastIdx := TO_DINT(THIS^.nCount - 1);
END_IF
END_GET
END_PROPERTY

PROPERTY PROTECTED pBuffer : POINTER TO I_Object
GET
pBuffer := THIS^.fbBuffer.pBuffer;
END_GET
END_PROPERTY

METHOD Remove : BOOL
VAR_INPUT
    ipObject:       I_Object;
END_VAR
VAR
    nIdxToRemove:   DINT;
END_VAR
IF ipObject = 0 THEN
    RETURN;
END_IF

nIdxToRemove := THIS^.IndexOfItem(ipObject);
Remove := THIS^.RemoveAt(nIdxToRemove);
END_METHOD

METHOD RemoveAt : BOOL
VAR_INPUT
    nIdx: DINT;
END_VAR
VAR
    nNewCapacity: UDINT;
END_VAR
IF NOT THIS^.IndexIsValid(nIdx)
    OR_ELSE THIS^.nCount = 0 THEN
    RETURN;
END_IF

THIS^.WriteToBuffer(nIdx := nIdx, ipObject := 0); // Reset memory at given idx

IF nIdx < THIS^.nLastIdx THEN
    Tc2_System.MEMMOVE(destAddr := THIS^.GetOffset(nIdx),
                       srcAddr := THIS^.GetOffset(nIdx + 1),
                       n := TO_UDINT(THIS^.nLastIdx - nIdx)*THIS^.nItemSize);
END_IF

THIS^._nCount := THIS^._nCount - 1;

IF THIS^.nCount*2 <= THIS^.nCapacity THEN
    nNewCapacity := MAX(Param_List.nDefaultCapacity, THIS^.nCount);

    IF nNewCapacity <> THIS^.nCapacity THEN
        THIS^.fbBuffer.Resize(nSize := nNewCapacity*THIS^.nItemSize,
                              bPreserve := TRUE,
                              bReset := FALSE);
    END_IF
END_IF

RemoveAt := TRUE;
END_METHOD

METHOD PUBLIC TrimCapacity
VAR_INPUT
END_VAR
THIS^.fbBuffer.Resize(nSize := THIS^.nCount*THIS^.nItemSize,
                      bPreserve := TRUE,
                      bReset := FALSE);
END_METHOD

METHOD PRIVATE WriteToBuffer : BOOL
VAR_INPUT
    nIdx: DINT;
    ipObject: I_Object;
END_VAR
VAR
    pTmp: POINTER TO I_Object;
END_VAR
IF NOT THIS^.IndexIsValid(nIdx) THEN
    RETURN;
END_IF

pTmp := THIS^.pBuffer;
pTmp[nIdx] := ipObject;
END_METHOD

END_FUNCTION_BLOCK

// ---- Helpers/F_CompareObjects.TcPOU
FUNCTION F_CompareObjects : BOOL
VAR_INPUT
    ipObject1:      I_Object;
    ipObject2:      I_Object;
END_VAR
VAR
END_VAR

IF ipObject1 = ipObject2 THEN
    F_CompareObjects := TRUE;
END_IF

END_FUNCTION

// ---- Action/Tests/FB_ActionTestObject.TcPOU
FUNCTION_BLOCK INTERNAL FB_ActionTestObject EXTENDS FB_Object IMPLEMENTS I_CyclicTask
VAR
    _nCounter: UDINT;
    _bActivated: BOOL;
END_VAR

METHOD Activate
VAR_INPUT
    bActivate: BOOL;
END_VAR
THIS^._bActivated := bActivate;
END_METHOD

PROPERTY bIsActivated : BOOL
GET
bIsActivated := THIS^._bActivated;
END_GET
END_PROPERTY

PROPERTY nCounter : UDINT
GET
nCounter := THIS^._nCounter;
END_GET
END_PROPERTY

METHOD Run
VAR_INPUT
END_VAR
THIS^._nCounter := THIS^._nCounter + 1;
END_METHOD

END_FUNCTION_BLOCK

// ---- Action/Tests/FB_ActivateAction.TcPOU
FUNCTION_BLOCK INTERNAL FB_ActivateAction EXTENDS FB_Action
VAR
    _bActivated: BOOL;
END_VAR

METHOD  Execute
VAR_INPUT
    ipObject: I_Object;
END_VAR
VAR
    p: POINTER TO FB_ActionTestObject;
END_VAR
__QUERYPOINTER(ipObject, p);

IF p <> 0 THEN
    p^.Activate(THIS^._bActivated);
END_IF
END_METHOD

METHOD Inputs : I_Action
VAR_INPUT
    bActivate: BOOL;
END_VAR
Inputs := THIS^;
THIS^._bActivated := bActivate;
END_METHOD

END_FUNCTION_BLOCK

// ---- Action/FB_Action.TcPOU
FUNCTION_BLOCK ABSTRACT FB_Action EXTENDS FB_Object IMPLEMENTS I_Action
VAR
END_VAR

METHOD ABSTRACT Execute
VAR_INPUT
    ipObject: I_Object;
END_VAR
END_METHOD

END_FUNCTION_BLOCK

// ---- Action/FB_RunCyclicTasksAction.TcPOU
FUNCTION_BLOCK FB_RunCyclicTasksAction EXTENDS FB_Action
VAR
END_VAR

METHOD  Execute
VAR_INPUT
    ipObject: I_Object;
END_VAR
VAR
    ipTask: I_CyclicTask;
END_VAR
IF __QUERYINTERFACE(ipObject, ipTask) THEN
    ipTask.Run();
END_IF
END_METHOD

END_FUNCTION_BLOCK

// ---- Collection/Tests/FB_ListCapacity_Test.TcPOU
FUNCTION_BLOCK INTERNAL FB_ListCapacity_Test EXTENDS TcUnit.FB_TestSuite
VAR_INPUT
END_VAR
VAR_OUTPUT
END_VAR
VAR
END_VAR

TestAddMoreItemsThanCurrentCapacityExpectCapacityToDouble();
TestInitializeCapacityWithNonZeroValuesExpectSuccess();
TestRemoveItemsLowerThanHalfCurrentCapacityExpectCapacityTrimmed();
TestTrimCapacityExpectCapacityEqualsCurrentItemCount();
TestTrimCapacityExpectTheSameContentsAsBefore();

METHOD PRIVATE TestAddMoreItemsThanCurrentCapacityExpectCapacityToDouble
VAR_INST
    fbList: FB_List(5);
    fbObject: FB_DummyObject;
    i: UDINT;
END_VAR
TcUnit.TEST('TestAddMoreItemsThanCurrentCapacityExpectCapacityToDouble');

THIS^.AssertEquals_UDINT(Expected := 5,
                         Actual := fbList.nCapacity,
                         Message := 'Unexpected initial capacity');

FOR i := 1 TO 21 DO
    fbList.AddItem(fbObject);
    IF 6 <= i AND_THEN i <= 10 THEN
        THIS^.AssertEquals_UDINT(Expected := 10,
                                 Actual := fbList.nCapacity,
                                 Message := 'Unexpected new capacity');
    ELSIF 10 < i AND_THEN i <= 11 THEN
        THIS^.AssertEquals_UDINT(Expected := 20,
                                 Actual := fbList.nCapacity,
                                 Message := 'Unexpected new capacity');
    ELSIF i > 20 THEN
        THIS^.AssertEquals_UDINT(Expected := 40,
                                 Actual := fbList.nCapacity,
                                 Message := 'Unexpected new capacity');
    END_IF
END_FOR


TcUnit.TEST_FINISHED();
END_METHOD

METHOD PRIVATE TestInitializeCapacityWithNonZeroValuesExpectSuccess
VAR_INST
    aList: ARRAY [1..5] OF FB_List[(4), (10), (20), (100), (1000)];
    aExpected: ARRAY [1..5] OF UDINT := [4, 10, 20, 100, 1000];
    i: UDINT;
END_VAR
TcUnit.TEST('TestInitializeCapacityWithNonZeroValuesExpectSuccess');

FOR i := 1 TO SIZEOF(aList)/SIZEOF(aList[1]) DO
    THIS^.AssertEquals_UDINT(Expected := aExpected[i],
                             Actual := aList[i].nCapacity,
                             Message := 'Unexpected capacity');
END_FOR

TcUnit.TEST_FINISHED();
END_METHOD

METHOD PRIVATE TestRemoveItemsLowerThanHalfCurrentCapacityExpectCapacityTrimmed
VAR_INST
    fbList: FB_List(5);
    fbObject: FB_DummyObject;
    i: UDINT;
END_VAR
TcUnit.TEST('TestRemoveItemsLowerThanHalfCurrentCapacityExpectCapacityTrimmed');

THIS^.AssertEquals_UDINT(Expected := 5,
                         Actual := fbList.nCapacity,
                         Message := 'Unexpected initial capacity');

FOR i := 1 TO 15 DO
    fbList.AddItem(fbObject);
END_FOR

THIS^.AssertEquals_UDINT(Expected := 20,
                         Actual := fbList.nCapacity,
                         Message := 'Unexpected new capacity');

FOR i := 1 TO 15 DO
    fbList.RemoveAt(0);
    IF 1 <= i AND_THEN i < 5 THEN
        THIS^.AssertEquals_UDINT(Expected := 20,
                                 Actual := fbList.nCapacity,
                                 Message := 'Capacity should not be reduced yet');
    ELSIF 5 <= i AND_THEN i < 10 THEN
        THIS^.AssertEquals_UDINT(Expected := 10,
                                 Actual := fbList.nCapacity,
                                 Message := 'Capacity should be trimmed');
    ELSIF 10 <= i AND_THEN i < 13 THEN
        THIS^.AssertEquals_UDINT(Expected := 5,
                                 Actual := fbList.nCapacity,
                                 Message := 'Capacity should be trimmed');
    ELSE
        THIS^.AssertEquals_UDINT(Expected := Param_List.nDefaultCapacity,
                                 Actual := fbList.nCapacity,
                                 Message := 'Capacity should not be lower than default capacity');
    END_IF
END_FOR

TcUnit.TEST_FINISHED();
END_METHOD

METHOD PRIVATE TestTrimCapacityExpectCapacityEqualsCurrentItemCount
VAR_INST
    fbList: FB_List(5);

    nTimesToAdd: UDINT;
    fbObject: FB_DummyObject;

    i: UDINT;
END_VAR
TcUnit.TEST('TestTrimCapacityExpectCapacityEqualsCurrentItemCount');

THIS^.AssertEquals_UDINT(Expected := 5,
                         Actual := fbList.nCapacity,
                         Message := 'Unexpected initial capacity');

nTimesToAdd := 6;

FOR i := 1 TO 15 DO
    fbList.AddItem(fbObject);
END_FOR

THIS^.AssertEquals_UDINT(Expected := 20,
                         Actual := fbList.nCapacity,
                         Message := 'Unexpected capacity before trimming');

fbList.TrimCapacity();

THIS^.AssertEquals_UDINT(Expected := 15,
                         Actual := fbList.nCapacity,
                         Message := 'Unexpected capacity after trimming');

TcUnit.TEST_FINISHED();
END_METHOD

METHOD PRIVATE TestTrimCapacityExpectTheSameContentsAsBefore
VAR_INST
    fbList: FB_List(5);

    nTimesToAdd: UDINT;
    fbObject: FB_DummyObject;

    i: UDINT;
END_VAR
TcUnit.TEST('TestTrimCapacityExpectTheSameContentsAsBefore');

THIS^.AssertEquals_UDINT(Expected := 5,
                         Actual := fbList.nCapacity,
                         Message := 'Unexpected initial capacity');

nTimesToAdd := 6;

FOR i := 1 TO 15 DO
    fbList.AddItem(fbObject);
END_FOR

THIS^.AssertEquals_UDINT(Expected := 20,
                         Actual := fbList.nCapacity,
                         Message := 'Unexpected capacity before trimming');

fbList.TrimCapacity();

THIS^.AssertEquals_UDINT(Expected := 15,
                         Actual := fbList.nCapacity,
                         Message := 'Unexpected capacity after trimming');

FOR i := 1 TO 15 DO
    THIS^.AssertTrue(Condition := fbList.ItemAt(TO_DINT(i - 1)).Equals(fbObject),
                     Message := CONCAT('Unexpected item at index ', TO_STRING(i)));
END_FOR

TcUnit.TEST_FINISHED();
END_METHOD

END_FUNCTION_BLOCK

// ---- Invocation Control/Tests/FB_InvocationControl_Test.TcPOU
FUNCTION_BLOCK INTERNAL FB_InvocationControl_Test EXTENDS TcUnit.FB_TestSuite
VAR
    
END_VAR

RunAllTheTimeExpectCalledCyclicallyTrue();
RunAllTheTimeExpectNewInvocationOnce();
RunOnceExpectNewInvocationOnce();
RunOncePerCycleExpectMultipleCallAlwaysFalse();
RunThricePerCycleExpectMultipleCallTrue();

METHOD PRIVATE RunAllTheTimeExpectCalledCyclicallyTrue
VAR_INST
    fbCallCtrl:             FB_InvocationControl;
    fbCallCtrlTestTask:     FB_InvocationControlTestTask;
END_VAR
TcUnit.TEST('RunAllTheTimeExpectCalledCyclicallyTrue');

fbCallCtrlTestTask.SetRunCondition(5).Run();

IF fbCallCtrlTestTask.nCycleCounter = 1 THEN
    THIS^.AssertFalse(Condition := fbCallCtrl.bCalledCyclically,
                      Message := '$'bCalledCyclically$' should be false as Track() has not been called at all');
END_IF

fbCallCtrl.Track();

THIS^.AssertTrue(Condition := fbCallCtrl.bCalledCyclically,
                 Message := '$'bCalledCyclically$' is false, but it should be true');

THIS^.AssertTrue(Condition := fbCallCtrl.bCalledThisCycle,
                 Message := '$'bCalledThisCycle$' is false, but it should be true');

IF fbCallCtrlTestTask.nCycleCounter > 1 THEN
    THIS^.AssertTrue(Condition := fbCallCtrl.bCalledLastCycle,
                     Message := '$'bCalledLastCycle$' is false, but it should be true');
    IF NOT fbCallCtrl.bCalledLastCycle THEN
        ADSLOGSTR(msgCtrlMask := ADSLOG_MSGTYPE_ERROR,
                  msgFmtStr := fbCallCtrl.ToString(),
                  strArg := '');
    END_IF
ELSE
    THIS^.AssertFalse(Condition := fbCallCtrl.bCalledLastCycle,
                      Message := '$'bCalledLastCycle$' should not be true on the first cycle it is called');
END_IF

IF fbCallCtrlTestTask.bDone THEN
    TcUnit.TEST_FINISHED();
END_IF
END_METHOD

METHOD PRIVATE RunAllTheTimeExpectNewInvocationOnce
VAR_INST
    fbCallCtrl:             FB_InvocationControl;
    fbCallCtrlTestTask:     FB_InvocationControlTestTask;
END_VAR
TcUnit.TEST('RunAllTheTimeExpectNewInvocationOnce');

fbCallCtrlTestTask.SetRunCondition(5).Run();

fbCallCtrl.Track();

IF fbCallCtrlTestTask.nCycleCounter = 1 THEN
    THIS^.AssertTrue(Condition := fbCallCtrl.bNewInvocation,
                     Message := '$'bNewInvocation$' is false, but it should be true');
ELSE
    THIS^.Assertfalse(Condition := fbCallCtrl.bNewInvocation,
                      Message := '$'bNewInvocation$' is true, but it should be false');
END_IF

IF fbCallCtrlTestTask.bDone THEN
    TcUnit.TEST_FINISHED();
END_IF
END_METHOD

METHOD PRIVATE RunOnceExpectNewInvocationOnce
VAR_INST
    fbCallCtrl:             FB_InvocationControl;
    fbCallCtrlTestTask:     FB_InvocationControlTestTask;
END_VAR
TcUnit.TEST('RunOnceExpectNewInvocationOnce');

fbCallCtrlTestTask.SetRunCondition(5).Run();

IF fbCallCtrlTestTask.nCycleCounter = 3 THEN
    fbCallCtrl.Track();
    THIS^.AssertTrue(Condition := fbCallCtrl.bNewInvocation,
                     Message := '$'bNewInvocation$' is false, but it should be true');
ELSE
    THIS^.AssertFalse(Condition := fbCallCtrl.bNewInvocation,
                      Message := '$'bNewInvocation$' is trie, but it should be false');
END_IF

IF fbCallCtrlTestTask.bDone THEN
    TcUnit.TEST_FINISHED();
END_IF
END_METHOD

METHOD PRIVATE RunOncePerCycleExpectMultipleCallAlwaysFalse
VAR_INST
    fbCallCtrl:             FB_InvocationControl;
    fbCallCtrlTestTask:     FB_InvocationControlTestTask;
END_VAR
TcUnit.TEST('RunOncePerCycleExpectMultipleCallAlwaysFalse');

fbCallCtrlTestTask.SetRunCondition(5).Run();

THIS^.AssertFalse(Condition := fbCallCtrl.bMultipleCall,
                  Message := '$'bMultipleCall$' is true, but it should be false');

fbCallCtrl.Track();

THIS^.AssertFalse(Condition := fbCallCtrl.bMultipleCall,
                  Message := '$'bMultipleCall$' is true, but it should be false');


IF fbCallCtrlTestTask.bDone THEN
    TcUnit.TEST_FINISHED();
END_IF
END_METHOD

METHOD PRIVATE RunThricePerCycleExpectMultipleCallTrue
VAR_INST
    fbCallCtrl:             FB_InvocationControl;
    fbCallCtrlTestTask:     FB_InvocationControlTestTask;
END_VAR
TcUnit.TEST('RunThricePerCycleExpectMultipleCallTrue');

fbCallCtrlTestTask.SetRunCondition(5).Run();

IF fbCallCtrlTestTask.nCycleCounter > 1 THEN
    THIS^.AssertTrue(Condition := fbCallCtrl.bMultipleCall,
                     Message := '$'bMultipleCall$' is false, but it should be true');
END_IF

fbCallCtrl.Track().Track().Track();

THIS^.AssertTrue(Condition := fbCallCtrl.bMultipleCall,
                 Message := '$'bMultipleCall$' is false, but it should be true');

IF fbCallCtrlTestTask.bDone THEN
    TcUnit.TEST_FINISHED();
END_IF
END_METHOD

END_FUNCTION_BLOCK

// ---- Invocation Control/FB_InvocationControl.TcPOU
{attribute 'reflection'}
FUNCTION_BLOCK FB_InvocationControl
// This FB can be used to track if a unit of code is executed cyclically or just invoked
// A unit of code can be, for example, the body of an FB, a method,
// an action, a property, etc.
//
// To track the desired task, simply place the Track() method in that task.
// Note that this FB can only track one unit of code at a time, and its properties
// must be used only after the Track() method is called.
VAR_INPUT
END_VAR
VAR_OUTPUT
END_VAR
VAR
    _sOutTemplate:              STRING(MAX_STRING_LENGTH);
    _sOut:                      STRING(MAX_STRING_LENGTH);
    fbGetCurTaskIdx:            GETCURTASKINDEX;
    _nTaskIdx:                  BYTE;
    _TaskId:                    OTCID;
    _nCycleCount:               UDINT; // Tracking cycle count
    _nOldCycleCount:            UDINT; // Old tracking cycle count
    _nCallCount:                UDINT; // Call count of Track()
    _nOldCallCount:             UDINT; // Old call count of Track()
    _nTaskTime:                 LINT;
    _nOldTaskTime:              LINT;
    {attribute 'instance-path'}
    {attribute 'noinit'}
    sPath:                      STRING(MAX_STRING_LENGTH);
END_VAR

PROPERTY bCalledCyclically : BOOL
GET
// New invocation when:
//      - 'Track()' was called last cycle, OR
//      - 'Track()' is called this cycle
bCalledCyclically := THIS^.TaskTracked() AND_THEN (THIS^.bCalledLastCycle OR_ELSE THIS^.bCalledThisCycle);
END_GET
END_PROPERTY

PROPERTY bCalledLastCycle : BOOL
GET
IF NOT THIS^.TaskTracked() THEN
    RETURN;
END_IF

IF THIS^.bCalledThisCycle THEN
    bCalledLastCycle := (THIS^.nOldCycleCount + 1) = THIS^.nTaskCycleCount;
ELSE
    bCalledLastCycle := (THIS^.nCycleCount + 1) = THIS^.nTaskCycleCount;
END_IF
END_GET
END_PROPERTY

PROPERTY bCalledThisCycle : BOOL
GET
bCalledThisCycle :=
    THIS^.TaskTracked() AND_THEN (THIS^.nCycleCount = THIS^.nTaskCycleCount);
END_GET
END_PROPERTY

PROPERTY bMultipleCall : BOOL
GET
// Multiple call when:
//  - 'TaskId' <> 0, and
//  - '_nOldCallCount' <> '_nOldCycleCount', and
//  - 'Track()' is called this cycle
bMultipleCall := THIS^.TaskTracked()
                 AND_THEN THIS^.bCalledCyclically
                 AND_THEN THIS^._nCallCount - THIS^._nOldCallCount > 1;
END_GET
END_PROPERTY

PROPERTY bNewInvocation : BOOL
GET
VAR_INST
    nLastTrigCycleCount:        UDINT;
END_VAR
// New invocation when:
//  - 'TaskId' <> 0, and
//  - 'Track()' was not called last cycle, and
//  - 'Track()' is called this cycle, and
bNewInvocation := THIS^.TaskTracked()
                  AND_THEN (THIS^.nOldCycleCount + 1) <> THIS^.nCycleCount
                  AND_THEN THIS^.nCycleCount = THIS^.nTaskCycleCount;

// For debugging
IF bNewInvocation THEN
    nLastTrigCycleCount := THIS^.nTaskCycleCount;
END_IF
END_GET
END_PROPERTY

METHOD FB_init : BOOL
VAR_INPUT
	bInitRetains : BOOL; // if TRUE, the retain variables are initialized (warm start / cold start)
	bInCopyCode : BOOL;  // if TRUE, the instance afterwards gets moved into the copy code (online change)
END_VAR
THIS^._sOutTemplate :=
        'TaskIdx=%d, 
         TaskId=%d, 
         TrackCycleCount=%d, 
         OldTrackCycleCount=%d, 
         TaskCycleCount=%d, 
         CallCount=%d, 
         OldCallCount=%d';
END_METHOD

PROPERTY nCycleCount : UDINT
GET
nCycleCount := THIS^._nCycleCount;
END_GET
END_PROPERTY

PROPERTY nOldCycleCount : UDINT
GET
nOldCycleCount := THIS^._nOldCycleCount;
END_GET
END_PROPERTY

PROPERTY nTaskCycleCount : UDINT
GET
IF THIS^.TaskTracked() THEN
    nTaskCycleCount := TwinCAT_SystemInfoVarList._TaskInfo[THIS^._nTaskIdx].CycleCount;
END_IF
END_GET
END_PROPERTY

METHOD PROTECTED TaskTracked : BOOL
VAR_INPUT
END_VAR
TaskTracked := THIS^._TaskId <> 0;
END_METHOD

METHOD ToString : STRING(MAX_STRING_LENGTH)
VAR_INST
    fbFormatStr:        FB_FormatString2;
END_VAR
fbFormatStr(pFormatString := ADR(THIS^._sOutTemplate),
            arg1 := F_BYTE(THIS^._nTaskIdx),
            arg2 := F_UDINT(THIS^._TaskId),
            arg3 := F_UDINT(THIS^._nCycleCount),
            arg4 := F_UDINT(THIS^._nOldCycleCount),
            arg5 := F_UDINT(TwinCAT_SystemInfoVarList._TaskInfo[THIS^._nTaskIdx].CycleCount),
            arg6 := F_UDINT(THIS^._nCallCount),
            arg7 := F_UDINT(THIS^._nOldCallCount),
            pDstString := ADR(THIS^._sOut),
            nDstSize := MAX_STRING_LENGTH);

ToString := THIS^._sOut;
END_METHOD

METHOD Track : REFERENCE TO FB_InvocationControl
VAR_INPUT
END_VAR
VAR
    nCurCycleCount:         UDINT;
END_VAR
Track REF= THIS^;

// Initialize '_TaskId'
IF THIS^._TaskId = 0 THEN
    THIS^.fbGetCurTaskIdx();
    THIS^._nTaskIdx := THIS^.fbGetCurTaskIdx.index;
    THIS^._TaskId := TwinCAT_SystemInfoVarList._TaskInfo[THIS^._nTaskIdx].ObjId;
END_IF

nCurCycleCount := THIS^.nTaskCycleCount;

// Update old info only if this is a new cycle
IF THIS^._nTaskTime <> TwinCAT_SystemInfoVarList._TaskInfo[THIS^._nTaskIdx].DcTaskTime THEN
    THIS^._nOldTaskTime := THIS^._nTaskTime;
    THIS^._nOldCycleCount := THIS^._nCycleCount;
    THIS^._nOldCallCount := THIS^._nCallCount;
ELSE
    THIS^._nCallCount := THIS^._nCallCount + 1;
END_IF

// Update current info
THIS^._nTaskTime := TwinCAT_SystemInfoVarList._TaskInfo[THIS^._nTaskIdx].DcTaskTime;
THIS^._nCycleCount := nCurCycleCount;
END_METHOD

END_FUNCTION_BLOCK

// ---- Invocation Control/Tests/FB_InvocationControlTestTask.TcPOU
FUNCTION_BLOCK INTERNAL FB_InvocationControlTestTask EXTENDS FB_Task
VAR CONSTANT
    cDefaultCyclesToRun:        UDINT := 1;
END_VAR
VAR
    _nCyclesToRunIn:            UDINT;

    _nCyclesToRun:              UDINT := 10;
    _nCycleCounter:             UDINT;
END_VAR

PROPERTY nCycleCounter : UDINT
GET
nCycleCounter := THIS^._nCycleCounter;
END_GET
END_PROPERTY

METHOD PROTECTED OnStart
VAR_INPUT
END_VAR
IF THIS^._nCyclesToRunIn > 0 THEN
    THIS^._nCyclesToRun := THIS^._nCyclesToRunIn;
ELSE
    THIS^._nCyclesToRun := THIS^.cDefaultCyclesToRun;
END_IF
END_METHOD

METHOD Restore : I_Restorable
Restore := SUPER^.Restore();

THIS^._nCycleCounter := 0;
END_METHOD

METHOD Run
VAR_INPUT
END_VAR
IF THIS^.Execute() THEN
    THIS^._nCycleCounter := THIS^._nCycleCounter + 1;

    THIS^.DoneWhen(THIS^._nCycleCounter = THIS^._nCyclesToRun);
END_IF
END_METHOD

METHOD SetRunCondition : REFERENCE TO FB_InvocationControlTestTask
VAR_INPUT
    nCyclesToRun:        UDINT; // Number of cycles to run
END_VAR
SetRunCondition REF= THIS^;

THIS^._nCyclesToRunIn := nCyclesToRun;

THIS^.Invoke();
END_METHOD

END_FUNCTION_BLOCK

// ---- Task/FB_Task.TcPOU
FUNCTION_BLOCK FB_Task EXTENDS FB_Object IMPLEMENTS I_Task, I_CyclicTask
VAR_INPUT
END_VAR
VAR_OUTPUT
END_VAR
VAR
    _eState:                E_TaskState;
    _eOldState:             E_TaskState;
    _nStartCounter:         UDINT := 0;
    fbExecutionTimer:       TON := (PT := TO_TIME(GVL_IntegerTypeBounds.DWORD_UPPER_BOUND));
    fbExecuteCallCtrl:      FB_InvocationControl;
END_VAR

METHOD Abort : I_TaskStatus
Abort := THIS^;

IF THIS^._eState = E_TaskState.Busy THEN
    THIS^.OnAbort();
    THIS^.Restore();
END_IF
END_METHOD

PROPERTY bBusy : BOOL
GET
bBusy := THIS^._eState = E_TaskState.Busy;
THIS^.CheckCyclicCall();
END_GET
END_PROPERTY

PROPERTY bDone : BOOL
GET
bDone := THIS^._eState = E_TaskState.Done;
THIS^.CheckCyclicCall();
END_GET
END_PROPERTY

PROPERTY bError : BOOL
GET
bError := THIS^._eState = E_TaskState.Error;
THIS^.CheckCyclicCall();
END_GET
END_PROPERTY

PROPERTY bReady : BOOL
GET
bReady := THIS^._eState = E_TaskState.Ready;
THIS^.CheckCyclicCall();
END_GET
END_PROPERTY

METHOD PRIVATE CheckCyclicCall
VAR_INST
    fbCallCtrl:             FB_InvocationControl;
END_VAR
fbCallCtrl.Track();

IF THIS^.eState = E_TaskState.Busy AND_THEN
    (THIS^.CyclicCallDropped()
        OR_ELSE (NOT THIS^.fbExecuteCallCtrl.bCalledCyclically AND_THEN fbCallCtrl.bNewInvocation)) THEN
    Tc2_System.ADSLOGSTR(
        msgCtrlMask := Tc2_System.ADSLOG_MSGTYPE_ERROR,
        msgFmtStr := 'Cyclic execution of is not done correctly for $'%s$'',
        strArg := THIS^.sPath);
END_IF
END_METHOD

METHOD PRIVATE CyclicCallDropped : BOOL
VAR_INST
    fbCyclicCallDropped:        F_TRIG;
END_VAR
fbCyclicCallDropped(CLK:= THIS^.fbExecuteCallCtrl.bCalledCyclically);

CyclicCallDropped := fbCyclicCallDropped.Q;
END_METHOD

METHOD DoneWhen : BOOL
VAR_INPUT
    bDone:          BOOL;
END_VAR
IF bDone AND_THEN THIS^._eState = E_TaskState.Busy THEN
    THIS^.SetState(E_TaskState.Done);
    THIS^.OnDone();
    DoneWhen := TRUE;
END_IF
END_METHOD

METHOD ErrorWhen : BOOL
VAR_INPUT
    bError:         BOOL;
END_VAR
IF bError AND_THEN THIS^._eState = E_TaskState.Busy THEN
    THIS^.SetState(E_TaskState.Error);
    THIS^.OnError();
    ErrorWhen := TRUE;
END_IF
END_METHOD

PROPERTY eState : E_TaskState
GET
eState := THIS^._eState;
END_GET
END_PROPERTY

METHOD PROTECTED Execute : BOOL
VAR_INPUT
END_VAR
THIS^.fbExecuteCallCtrl.Track();

IF THIS^._eState = E_TaskState.Error THEN
    THIS^.WhileError();
END_IF;

Execute := THIS^._eState = E_TaskState.Busy;

IF Execute THEN
    THIS^.fbExecutionTimer(IN := TRUE);
END_IF
END_METHOD

METHOD Invoke : I_TaskStatus
VAR_INST
    fbCallCtrl:         FB_InvocationControl;
END_VAR
fbCallCtrl.Track();

IF THIS^._eState = E_TaskState.Ready
    OR_ELSE ((THIS^._eState = E_TaskState.Done OR THIS^._eState = E_TaskState.Error) AND fbCallCtrl.bNewInvocation) THEN

    THIS^.SetState(E_TaskState.Busy);
    THIS^._nStartCounter := THIS^._nStartCounter + 1;
    THIS^.fbExecutionTimer(IN := FALSE);
    THIS^.OnStart();
END_IF

Invoke := THIS^;
END_METHOD

METHOD PROTECTED OnAbort
VAR_INPUT
END_VAR
END_METHOD

METHOD PROTECTED OnDone
VAR_INPUT
END_VAR
END_METHOD

METHOD PROTECTED OnError
VAR_INPUT
END_VAR
END_METHOD

METHOD PROTECTED OnStart
VAR_INPUT
END_VAR
END_METHOD

METHOD Restore : I_Restorable
THIS^.SetState(E_TaskState.Ready);
THIS^.fbExecutionTimer(IN := FALSE);

Restore := THIS^;
END_METHOD

METHOD Run
VAR_INPUT
END_VAR
END_METHOD

METHOD PRIVATE SetState
VAR_INPUT
    eNewState:          E_TaskState;
END_VAR
IF THIS^._eState <> eNewState THEN
    THIS^._eOldState := THIS^._eState;
    THIS^._eState := eNewState;
END_IF
END_METHOD

PROPERTY tElapsedTime : TIME
GET
tElapsedTime := fbExecutionTimer.ET;
END_GET
END_PROPERTY

METHOD PROTECTED WhileError
VAR_INPUT
END_VAR
END_METHOD

END_FUNCTION_BLOCK

// ---- Observer Pattern/Tests/FB_ObserverPattern_Test.TcPOU
FUNCTION_BLOCK INTERNAL FB_ObserverPattern_Test EXTENDS TcUnit.FB_TestSuite
// All observable types implements the same base methods for
// managing the list of observers, hence testing only one type
// of observable is enough. For instance, methods like, `Attach`,
// and `Detach`.
VAR
    fVal: LREAL;
END_VAR

TestAdd5CompatibleObserversExpectAll5();
TestAdd6IncompatibleObserversExpectNone();
TestAddDuplicateObserversExpectFailure();
TestAddNullObserverExpectFailure();
TestClearAllObserversExpectSuccess();
TestCompatibleDataTypesExpectValuesToUpdate();
TestDataTypeConsistencyOfObservables();
TestDataTypeConsistencyOfObservers();
TestDetachAddedObserversExpectSuccess();
TestExternalWithCompatibleDataTypeExpectValueToUpdate();
TestIncompatileDataTypesExpectNoValueChange();
TestNotifyAlwaysUponWriteAccess();
TestNotifyOnlyWhenValueChanged();
TestNotifyUponAttachmentWithObservers();
TestOneObservableToManyObserversExpectAllToUpdateValueAccordingly();

METHOD PRIVATE TestAdd5CompatibleObserversExpectAll5
VAR_INST
    fbObservableReal: FB_Observable_REAL;
    aObserverReal: ARRAY [1..5] OF FB_Observer_REAL;

    i: UDINT;
END_VAR
TcUnit.TEST('TestAdd5CompatibleObserversExpectAll5');

FOR i := 1 TO SIZEOF(aObserverReal)/SIZEOF(aObserverReal[1]) DO
    THIS^.AssertTrue(Condition := fbObservableReal.Attach(aObserverReal[i]),
                     Message := 'Failed to add compatible observer to observable');
END_FOR

THIS^.AssertEquals_UDINT(Expected := 5,
                         Actual := fbObservableReal.nObserverCount,
                         Message := 'Unexpected number of observers attached');

TcUnit.TEST_FINISHED();
END_METHOD

METHOD PRIVATE TestAdd6IncompatibleObserversExpectNone
VAR_INST
    // Test can be less manual with dynamic list
    fbObservableDint: FB_Observable_DINT;
    fbObservableUdint: FB_Observable_UDINT;
    fbObservableUint: FB_Observable_UINT;
    fbObservableReal: FB_Observable_REAL;
    fbObservableLreal: FB_Observable_LREAL;

    fbObserverDint: ARRAY [1..6] OF FB_Observer_DINT;
    fbObserverUdint: ARRAY [1..6] OF FB_Observer_UDINT;
    fbObserverUint: ARRAY [1..6] OF FB_Observer_UINT;
    fbObserverLreal: ARRAY [1..6] OF FB_Observer_LREAL;
    fbObserverReal: ARRAY [1..6] OF FB_Observer_REAL;

    i: UDINT;
END_VAR
TcUnit.TEST('TestAdd6IncompatibleObserversExpectNone');

FOR i := 1 TO SIZEOF(fbObserverUdint)/SIZEOF(fbObserverUdint[1]) DO
    fbObservableDint.Attach(fbObserverUdint[i]);
    fbObservableDint.Attach(fbObserverUint[i]);
    fbObservableDint.Attach(fbObserverLreal[i]);
    fbObservableDint.Attach(fbObserverReal[i]);

    fbObservableUdint.Attach(fbObserverDint[i]);
    fbObservableUdint.Attach(fbObserverUint[i]);
    fbObservableUdint.Attach(fbObserverLreal[i]);
    fbObservableUdint.Attach(fbObserverReal[i]);

    fbObservableUint.Attach(fbObserverDint[i]);
    fbObservableUint.Attach(fbObserverUdint[i]);
    fbObservableUint.Attach(fbObserverLreal[i]);
    fbObservableUint.Attach(fbObserverReal[i]);

    fbObservableLreal.Attach(fbObserverDint[i]);
    fbObservableLreal.Attach(fbObserverUdint[i]);
    fbObservableLreal.Attach(fbObserverUint[i]);
    fbObservableLreal.Attach(fbObserverReal[i]);

    fbObservableReal.Attach(fbObserverDint[i]);
    fbObservableReal.Attach(fbObserverUdint[i]);
    fbObservableReal.Attach(fbObserverUint[i]);
    fbObservableReal.Attach(fbObserverLreal[i]);

END_FOR

THIS^.AssertEquals_UDINT(Expected := 0,
                         Actual := fbObservableDint.nObserverCount,
                         Message := 'Unexpected number of observers attached to observable type DINT');

THIS^.AssertEquals_UDINT(Expected := 0,
                         Actual := fbObservableUdint.nObserverCount,
                         Message := 'Unexpected number of observers attached to observable type UDINT');

THIS^.AssertEquals_UDINT(Expected := 0,
                         Actual := fbObservableUint.nObserverCount,
                         Message := 'Unexpected number of observers attached to observable type UINT');

THIS^.AssertEquals_UDINT(Expected := 0,
                         Actual := fbObservableLreal.nObserverCount,
                         Message := 'Unexpected number of observers attached to observable type LREAL');

THIS^.AssertEquals_UDINT(Expected := 0,
                         Actual := fbObservableReal.nObserverCount,
                         Message := 'Unexpected number of observers attached to observable type REAL');

TcUnit.TEST_FINISHED();
END_METHOD

METHOD PRIVATE TestAddDuplicateObserversExpectFailure
VAR_INST
    fbObservableReal: FB_Observable_REAL;

    fbObserverReal: FB_Observer_REAL;

    i: UDINT;
END_VAR
TcUnit.TEST('TestAddDuplicateObserversExpectFailure');

FOR i := 1 TO 5 DO
    IF i = 1 THEN
        THIS^.AssertTrue(Condition := fbObservableReal.Attach(fbObserverReal),
                         Message := 'Failed to add compatible observer to observable');
    ELSE
        THIS^.AssertFalse(Condition := fbObservableReal.Attach(fbObserverReal),
                          Message := 'Observable should not add duplicate observers');
    END_IF
END_FOR

THIS^.AssertEquals_UDINT(Expected := 1,
                         Actual := fbObservableReal.nObserverCount,
                         Message := 'Unexpected number of observers attached');

TcUnit.TEST_FINISHED();
END_METHOD

METHOD PRIVATE TestAddNullObserverExpectFailure
VAR_INST
    ipNullObs: I_Observer;
    fbObservable: FB_Observable_LREAL;
END_VAR
TcUnit.TEST('TestAddNullObserverExpectFailure');

fbObservable.Attach(ipNullObs);

THIS^.AssertEquals_UDINT(Expected := 0,
                         Actual := fbObservable.nObserverCount,
                         Message := 'Invalid observer added');

TcUnit.TEST_FINISHED();
END_METHOD

METHOD PRIVATE TestClearAllObserversExpectSuccess
VAR_INST
    fbObservableReal: FB_Observable_REAL;
    aObserverReal: ARRAY [1..5] OF FB_Observer_REAL;

    i: UDINT;
END_VAR
TcUnit.TEST('TestClearAllObserversExpectSuccess');

FOR i := 1 TO SIZEOF(aObserverReal)/SIZEOF(aObserverReal[1]) DO
    fbObservableReal.Attach(aObserverReal[i]);
END_FOR

fbObservableReal.ClearAll();

THIS^.AssertEquals_UDINT(Expected := 0,
                         Actual := fbObservableReal.nObserverCount,
                         Message := 'Failed to clear all observers');

TcUnit.TEST_FINISHED();
END_METHOD

METHOD PRIVATE TestCompatibleDataTypesExpectValuesToUpdate
VAR_INST
    fbObservableBool: FB_Observable_BOOL;
    fbObservableByte: FB_Observable_BYTE;
    fbObservableWord: FB_Observable_WORD;
    fbObservableDword: FB_Observable_DWORD;
    fbObservableLword: FB_Observable_LWORD;
    fbObservableSint: FB_Observable_SINT;
    fbObservableUsint: FB_Observable_USINT;
    fbObservableInt: FB_Observable_INT;
    fbObservableUint: FB_Observable_UINT;
    fbObservableDint: FB_Observable_DINT;
    fbObservableUdint: FB_Observable_UDINT;
    fbObservableLint: FB_Observable_LINT;
    fbObservableUlint: FB_Observable_ULINT;
    fbObservableLreal: FB_Observable_LREAL;
    fbObservableReal: FB_Observable_REAL;

    fbObserverBool: FB_Observer_BOOL;
    fbObserverByte: FB_Observer_BYTE;
    fbObserverWord: FB_Observer_WORD;
    fbObserverDword: FB_Observer_DWORD;
    fbObserverLword: FB_Observer_LWORD;
    fbObserverSint: FB_Observer_SINT;
    fbObserverUsint: FB_Observer_USINT;
    fbObserverInt: FB_Observer_INT;
    fbObserverUint: FB_Observer_UINT;
    fbObserverDint: FB_Observer_DINT;
    fbObserverUdint: FB_Observer_UDINT;
    fbObserverLint: FB_Observer_LINT;
    fbObserverUlint: FB_Observer_ULINT;
    fbObserverLreal: FB_Observer_LREAL;
    fbObserverReal: FB_Observer_REAL;

    bVal: BOOL;
    i: UDINT;
END_VAR
TcUnit.TEST('TestCompatibleDataTypesExpectValuesToUpdate');

fbObservableBool.Attach(fbObserverBool);
fbObservableByte.Attach(fbObserverByte);
fbObservableWord.Attach(fbObserverWord);
fbObservableDword.Attach(fbObserverDword);
fbObservableLword.Attach(fbObserverLword);
fbObservableSint.Attach(fbObserverSint);
fbObservableUsint.Attach(fbObserverUsint);
fbObservableUint.Attach(fbObserverUint);
fbObservableInt.Attach(fbObserverInt);
fbObservableDint.Attach(fbObserverDint);
fbObservableUdint.Attach(fbObserverUdint);
fbObservableLint.Attach(fbObserverLint);
fbObservableUlint.Attach(fbObserverUlint);
fbObservableLreal.Attach(fbObserverLreal);
fbObservableReal.Attach(fbObserverReal);

FOR i := 1 TO 10 DO
    bVal := NOT bVal;
    fbObservableBool.bVal := bVal;
    fbObservableByte.nValue8 := TO_BYTE(i);
    fbObservableWord.nValue16 := TO_WORD(i);
    fbObservableDword.nValue32 := TO_DWORD(i);
    fbObservableLword.nValue64 := TO_LWORD(i);
    fbObservableSint.nValue8 := TO_SINT(i);
    fbObservableUsint.nValue8 := TO_USINT(i);
    fbObservableInt.nValue16 := TO_INT(i);
    fbObservableUint.nValue16 := TO_UINT(i);
    fbObservableDint.nValue32 := TO_DINT(i);
    fbObservableUdint.nValue32 := i;
    fbObservableLint.nValue64 := TO_LINT(i);
    fbObservableUlint.nValue64 := TO_ULINT(i);
    fbObservableLreal.fValue64 := TO_LREAL(i);
    fbObservableReal.fValue32 := TO_REAL(i);

    THIS^.AssertEquals_BOOL(Expected := bVal,
                            Actual := fbObserverBool.bValue,
                            Message := 'BOOL observer failed to update value according to observable');
    THIS^.AssertEquals_BYTE(Expected := TO_BYTE(i),
                            Actual := fbObserverByte.nValue8,
                            Message := 'BYTE observer failed to update value according to observable');
    THIS^.AssertEquals_WORD(Expected := TO_WORD(i),
                            Actual := fbObserverWord.nValue16,
                            Message := 'WORD observer failed to update value according to observable');
    THIS^.AssertEquals_DWORD(Expected := TO_DWORD(i),
                             Actual := fbObserverDword.nValue32,
                             Message := 'DWORD observer failed to update value according to observable');
    THIS^.AssertEquals_LWORD(Expected := TO_LWORD(i),
                             Actual := fbObserverLword.nValue64,
                             Message := 'LWORD observer failed to update value according to observable');
    THIS^.AssertEquals_SINT(Expected := TO_SINT(i),
                            Actual := fbObserverSint.nValue8,
                            Message := 'SINT observer failed to update value according to observable');
    THIS^.AssertEquals_USINT(Expected := TO_USINT(i),
                             Actual := fbObserverUsint.nValue8,
                             Message := 'USINT observer failed to update value according to observable');
    THIS^.AssertEquals_INT(Expected := TO_INT(i),
                           Actual := fbObserverInt.nValue16,
                           Message := 'INT observer failed to update value according to observable');
    THIS^.AssertEquals_UINT(Expected := TO_UINT(i),
                            Actual := fbObserverUint.nValue16,
                            Message := 'UINT observer failed to update value according to observable');
    THIS^.AssertEquals_DINT(Expected := TO_DINT(i),
                            Actual := fbObserverDint.nValue32,
                            Message := 'DINT observer failed to update value according to observable');
    THIS^.AssertEquals_UDINT(Expected := i,
                             Actual := fbObserverUdint.nValue32,
                             Message := 'UDINT observer failed to update value according to observable');
    THIS^.AssertEquals_LINT(Expected := TO_LINT(i),
                            Actual := fbObserverLint.nValue64,
                            Message := 'LINT observer failed to update value according to observable');
    THIS^.AssertEquals_LREAL(Expected := TO_LREAL(i),
                             Actual := fbObserverLreal.fValue64,
                             Delta := 0.01,
                             Message := 'LREAL observer failed to update value according to observable');
    THIS^.AssertEquals_REAL(Expected := TO_REAL(i),
                            Actual := fbObserverReal.fValue32,
                            Delta := 0.01,
                            Message := 'REAL observer failed to update value according to observable');
END_FOR

TcUnit.TEST_FINISHED();
END_METHOD

METHOD PRIVATE TestDataTypeConsistencyOfObservables
VAR_INST
    aTypes: ARRAY [1..15] OF __SYSTEM.TYPE_CLASS :=
        [
            __SYSTEM.TYPE_CLASS.TYPE_BOOL,
            __SYSTEM.TYPE_CLASS.TYPE_BYTE,
            __SYSTEM.TYPE_CLASS.TYPE_WORD,
            __SYSTEM.TYPE_CLASS.TYPE_DWORD,
            __SYSTEM.TYPE_CLASS.TYPE_LWORD,
            __SYSTEM.TYPE_CLASS.TYPE_SINT,
            __SYSTEM.TYPE_CLASS.TYPE_USINT,
            __SYSTEM.TYPE_CLASS.TYPE_INT,
            __SYSTEM.TYPE_CLASS.TYPE_UINT,
            __SYSTEM.TYPE_CLASS.TYPE_DINT,
            __SYSTEM.TYPE_CLASS.TYPE_UDINT,
            __SYSTEM.TYPE_CLASS.TYPE_LINT,
            __SYSTEM.TYPE_CLASS.TYPE_ULINT,
            __SYSTEM.TYPE_CLASS.TYPE_LREAL,
            __SYSTEM.TYPE_CLASS.TYPE_REAL
        ];

    fbList: FB_List(0);
    fbObservableBool: FB_Observable_BOOL;
    fbObservableByte: FB_Observable_BYTE;
    fbObservableWord: FB_Observable_WORD;
    fbObservableDword: FB_Observable_DWORD;
    fbObservableLword: FB_Observable_LWORD;
    fbObservableSint: FB_Observable_SINT;
    fbObservableUsint: FB_Observable_USINT;
    fbObservableInt: FB_Observable_INT;
    fbObservableUint: FB_Observable_UINT;
    fbObservableDint: FB_Observable_DINT;
    fbObservableUdint: FB_Observable_UDINT;
    fbObservableLint: FB_Observable_LINT;
    fbObservableUlint: FB_Observable_ULINT;
    fbObservableLreal: FB_Observable_LREAL;
    fbObservableReal: FB_Observable_REAL;

    ipTmp: I_Observable;
    i: UDINT;
END_VAR
TcUnit.TEST('TestExpectConsistentDataTypeOfObservables');

fbList.AddItem(fbObservableBool);
fbList.AddItem(fbObservableByte);
fbList.AddItem(fbObservableWord);
fbList.AddItem(fbObservableDword);
fbList.AddItem(fbObservableLword);
fbList.AddItem(fbObservableSint);
fbList.AddItem(fbObservableUsint);
fbList.AddItem(fbObservableInt);
fbList.AddItem(fbObservableUint);
fbList.AddItem(fbObservableDint);
fbList.AddItem(fbObservableUdint);
fbList.AddItem(fbObservableLint);
fbList.AddItem(fbObservableUlint);
fbList.AddItem(fbObservableLreal);
fbList.AddItem(fbObservableReal);

FOR i := 1 TO SIZEOF(aTypes)/SIZEOF(aTypes[i]) DO
    __QUERYINTERFACE(fbList.ItemAt(TO_DINT(i - 1)), ipTmp);
    THIS^.AssertEquals_UDINT(Expected := aTypes[i],
                             Actual := ipTmp.nTypeClass,
                             Message := CONCAT('Inconsistent type class for observable tested at index ', TO_STRING(i)));
END_FOR

TcUnit.TEST_FINISHED();
END_METHOD

METHOD PRIVATE TestDataTypeConsistencyOfObservers
VAR_INST
    aTypes: ARRAY [1..15] OF __SYSTEM.TYPE_CLASS :=
        [
            __SYSTEM.TYPE_CLASS.TYPE_BOOL,
            __SYSTEM.TYPE_CLASS.TYPE_BYTE,
            __SYSTEM.TYPE_CLASS.TYPE_WORD,
            __SYSTEM.TYPE_CLASS.TYPE_DWORD,
            __SYSTEM.TYPE_CLASS.TYPE_LWORD,
            __SYSTEM.TYPE_CLASS.TYPE_SINT,
            __SYSTEM.TYPE_CLASS.TYPE_USINT,
            __SYSTEM.TYPE_CLASS.TYPE_INT,
            __SYSTEM.TYPE_CLASS.TYPE_UINT,
            __SYSTEM.TYPE_CLASS.TYPE_DINT,
            __SYSTEM.TYPE_CLASS.TYPE_UDINT,
            __SYSTEM.TYPE_CLASS.TYPE_LINT,
            __SYSTEM.TYPE_CLASS.TYPE_ULINT,
            __SYSTEM.TYPE_CLASS.TYPE_LREAL,
            __SYSTEM.TYPE_CLASS.TYPE_REAL
        ];

    fbList: FB_List(0);
    fbObserverBool: FB_Observer_BOOL;
    fbObserverByte: FB_Observer_BYTE;
    fbObserverWord: FB_Observer_WORD;
    fbObserverDword: FB_Observer_DWORD;
    fbObserverLword: FB_Observer_LWORD;
    fbObserverSint: FB_Observer_SINT;
    fbObserverUsint: FB_Observer_USINT;
    fbObserverInt: FB_Observer_INT;
    fbObserverUint: FB_Observer_UINT;
    fbObserverDint: FB_Observer_DINT;
    fbObserverUdint: FB_Observer_UDINT;
    fbObserverLint: FB_Observer_LINT;
    fbObserverUlint: FB_Observer_ULINT;
    fbObserverLreal: FB_Observer_LREAL;
    fbObserverReal: FB_Observer_REAL;

    ipTmp: I_Observer;
    i: UDINT;
END_VAR
TcUnit.TEST('TestExpectConsistentDataTypeOfObservers');

fbList.AddItem(fbObserverBool);
fbList.AddItem(fbObserverByte);
fbList.AddItem(fbObserverWord);
fbList.AddItem(fbObserverDword);
fbList.AddItem(fbObserverLword);
fbList.AddItem(fbObserverSint);
fbList.AddItem(fbObserverUsint);
fbList.AddItem(fbObserverInt);
fbList.AddItem(fbObserverUint);
fbList.AddItem(fbObserverDint);
fbList.AddItem(fbObserverUdint);
fbList.AddItem(fbObserverLint);
fbList.AddItem(fbObserverUlint);
fbList.AddItem(fbObserverLreal);
fbList.AddItem(fbObserverReal);

FOR i := 1 TO SIZEOF(aTypes)/SIZEOF(aTypes[i]) DO
    __QUERYINTERFACE(fbList.ItemAt(TO_DINT(i - 1)), ipTmp);
    THIS^.AssertEquals_UDINT(Expected := aTypes[i],
                             Actual := ipTmp.nTypeClass,
                             Message := CONCAT('Inconsistent type class for observable tested at index ', TO_STRING(i)));
END_FOR

TcUnit.TEST_FINISHED();
END_METHOD

METHOD PRIVATE TestDetachAddedObserversExpectSuccess
VAR_INST
    fbObservableReal: FB_Observable_REAL;
    fbObserverReal: ARRAY [1..5] OF FB_Observer_REAL;

    i: UDINT;
END_VAR
TcUnit.TEST('TestDetachAddedObserversExpectSuccess');

FOR i := 1 TO SIZEOF(fbObserverReal)/SIZEOF(fbObserverReal[1]) DO
    fbObservableReal.Attach(fbObserverReal[i]);
END_FOR

FOR i := 1 TO SIZEOF(fbObserverReal)/SIZEOF(fbObserverReal[1]) DO
    THIS^.AssertTrue(Condition := fbObservableReal.Detach(fbObserverReal[i]),
                     Message := 'Failed to deatch added observer');

END_FOR

THIS^.AssertEquals_UDINT(Expected := 0,
                         Actual := fbObservableReal.nObserverCount,
                         Message := 'Unexpected number of observers attached');

TcUnit.TEST_FINISHED();
END_METHOD

METHOD PRIVATE TestExternalWithCompatibleDataTypeExpectValueToUpdate
VAR_INST
    fbObservableLreal: FB_Observable_LREAL;
    fbObserverExt: FB_ObserverExt(THIS^.fVal);
    aTestVal: ARRAY [1..5] OF LREAL :=
        [2.7183, 3.1415, -1, 1.6180, 6.6261];
    i: UDINT;
END_VAR
TcUnit.TEST('TestObserverExternalWithCompatibleDataTypeExpectValueToUpdate');

fbObservableLreal.Attach(fbObserverExt);

FOR i := 1 TO SIZEOF(aTestVal)/SIZEOF(aTestVal[1]) DO
    fbObservableLreal.fValue64 := aTestVal[i];
    THIS^.AssertEquals_LREAL(Expected := aTestVal[i],
                             Actual := THIS^.fVal,
                             Delta := 0.001,
                             Message := 'External observer typed LREAL failed to update value according to observable');
END_FOR

TcUnit.TEST_FINISHED();
END_METHOD

METHOD PRIVATE TestIncompatileDataTypesExpectNoValueChange
VAR_INST
    fbObservableReal: FB_Observable_REAL;

    fbObserverDint: FB_Observer_DINT;
    fbObserverUdint: FB_Observer_UDINT;
    fbObserverUint: FB_Observer_UINT;
    fbObserverLreal: FB_Observer_LREAL;

    i: UDINT;
END_VAR
TcUnit.TEST('TestIncompatileDataTypeObserverAndObservableExpectNoValueChange');

fbObservableReal.Attach(fbObserverDint);
fbObservableReal.Attach(fbObserverUdint);
fbObservableReal.Attach(fbObserverUint);
fbObservableReal.Attach(fbObserverLreal);

FOR i := 1 TO 10 DO
    fbObservableReal.fValue32 := TO_REAL(i);

    THIS^.AssertEquals_DINT(Expected := 0,
                            Actual := fbObserverDint.nValue32,
                            Message := 'DINT observer value is not 0, but it should be 0');

    THIS^.AssertEquals_UDINT(Expected := 0,
                            Actual := fbObserverUdint.nValue32,
                            Message := 'UDINT observer value is not 0, but it should be 0');

    THIS^.AssertEquals_UINT(Expected := 0,
                            Actual := fbObserverUint.nValue16,
                            Message := 'UINT observer value is not 0, but it should be 0');

    THIS^.AssertEquals_LREAL(Expected := 0,
                             Actual := fbObserverLreal.fValue64,
                             Delta := 0.001,
                             Message := 'LREAL observer value is not 0, but it should be 0');
END_FOR

TcUnit.TEST_FINISHED();
END_METHOD

METHOD PRIVATE TestNotifyAlwaysUponWriteAccess
VAR_INST
    fbObservable: FB_Observable_LREAL;
    fbObserver: FB_Observer_LREAL_;

    i: UDINT;
END_VAR
TcUnit.TEST('TestNotifyAlwaysUponWriteAccess');

fbObservable.bNotifyWhenChanged := FALSE;
fbObservable.Attach(fbObserver);

// Expect 1 update already because observable always update its observer upon
// attachment
THIS^.AssertEquals_UDINT(Expected := 1,
                         Actual := fbObserver.nUpdateCounter,
                         Message := 'Unexpected number of updates to observer');

FOR i := 1 TO 5 DO
    fbObservable.fValue64 := 1.0;
END_FOR

THIS^.AssertEquals_UDINT(Expected := 6,
                         Actual := fbObserver.nUpdateCounter,
                         Message := 'Unexpected number of updates to observer');

TcUnit.TEST_FINISHED();
END_METHOD

METHOD PRIVATE TestNotifyOnlyWhenValueChanged
VAR_INST
    fbObservable: FB_Observable_LREAL;
    fbObserver: FB_Observer_LREAL_;
    aVal: ARRAY [1..5] OF LREAL :=
        [2.7183, 3.1415, -1, 1.6180, 6.6261];

    i: UDINT;
    j: UDINT;
END_VAR
TcUnit.TEST('TestNotifyOnlyWhenValueChanged');

fbObservable.bNotifyWhenChanged := TRUE;
fbObservable.Attach(fbObserver);

// Expect 1 update already because observable always update its observer upon
// attachment
THIS^.AssertEquals_UDINT(Expected := 1,
                         Actual := fbObserver.nUpdateCounter,
                         Message := 'Unexpected number of updates to observer');

FOR i := 1 TO SIZEOF(aVal)/SIZEOF(aVal[1]) DO
    FOR j := 1 TO 5 DO
        fbObservable.fValue64 := aVal[i];
    END_FOR

    THIS^.AssertEquals_UDINT(Expected := i + 1,
                             Actual := fbObserver.nUpdateCounter,
                             Message := 'Unexpected number of updates to observer');
END_FOR


TcUnit.TEST_FINISHED();
END_METHOD

METHOD PRIVATE TestNotifyUponAttachmentWithObservers
VAR_INST
    fbObservable: FB_Observable_LREAL;
    aObserver: ARRAY [1..5] OF FB_Observer_LREAL_;

    i: UDINT;
END_VAR
TcUnit.TEST('TestNotifyUponAttachmentWithObservers');

fbObservable.fValue64 := 100.0;

FOR i := 1 TO SIZEOF(aObserver)/SIZEOF(aObserver[1]) DO
    fbObservable.Attach(aObserver[i]);
END_FOR

FOR i := 1 TO SIZEOF(aObserver)/SIZEOF(aObserver[1]) DO
    THIS^.AssertEquals_LREAL(Expected := fbObservable.fValue64,
                             Actual := aObserver[i].fValue64,
                             Delta := 0.01,
                             Message := 'Observer$'s value is not matching its observable upon attachment');
    THIS^.AssertEquals_UDINT(Expected := 1,
                             Actual := aObserver[i].nUpdateCounter,
                             Message := 'Unexpected number of updates to observer');
END_FOR

TcUnit.TEST_FINISHED();
END_METHOD

METHOD PRIVATE TestOneObservableToManyObserversExpectAllToUpdateValueAccordingly
VAR_INST
    fbObservableLreal: FB_Observable_LREAL;
    aObservers: ARRAY [1..5] OF FB_Observer_LREAL;
    aTestVal: ARRAY [1..5] OF LREAL :=
        [2.7183, 3.1415, -1, 1.6180, 6.6261];
    i: UDINT;
    j: UDINT;
END_VAR
TcUnit.TEST('TestOneObservableToManyObserversExpectAllToUpdateValueAccordingly');

FOR i := 1 TO SIZEOF(aObservers)/SIZEOF(aObservers[1]) DO
    fbObservableLreal.Attach(aObservers[i]);
END_FOR

FOR i := 1 TO SIZEOF(aTestVal)/SIZEOF(aTestVal[1]) DO
    fbObservableLreal.fValue64 := aTestVal[i];
    FOR j := 1 TO SIZEOF(aObservers)/SIZEOF(aObservers[1]) DO
        THIS^.AssertEquals_LREAL(Expected := aTestVal[i],
                         Actual := aObservers[j].fValue64,
                         Delta := 0.001,
                         Message := ' typed LREAL failed to update value according to observable');
    END_FOR
END_FOR

TcUnit.TEST_FINISHED();
END_METHOD

END_FUNCTION_BLOCK

// ---- Observer Pattern/FB_Observable_REAL.TcPOU
FUNCTION_BLOCK FB_Observable_REAL EXTENDS FB_AbstractObservable
VAR
    _fVal:                  REAL;
    _fOldVal:               LREAL;
END_VAR

METHOD FB_init : BOOL
VAR_INPUT
    bInitRetains:       BOOL; // if TRUE, the retain variables are initialized (warm start / cold start)
    bInCopyCode:        BOOL;  // if TRUE, the instance afterwards gets moved into the copy code (online change)
END_VAR
THIS^._nTypeClass := __SYSTEM.TYPE_CLASS.TYPE_REAL;
END_METHOD

PROPERTY fValue32 : REAL
GET
fValue32 := THIS^._fVal;
END_GET
SET
THIS^._fOldVal := _fVal;
THIS^._fVal := fValue32;

THIS^.NotifyWithConditions();
END_SET
END_PROPERTY

PROPERTY nDataSize : UDINT
GET
nDataSize := SIZEOF(REAL);
END_GET
END_PROPERTY

PROPERTY PROTECTED pData : POINTER TO BYTE
GET
pData := ADR(THIS^._fVal);
END_GET
END_PROPERTY

METHOD  ValueChanged : BOOL
VAR_INPUT
END_VAR
ValueChanged := THIS^._fOldVal <> THIS^._fVal;
END_METHOD

